LIN {X 0,Y 108.125,Z 394.279,A -85,B 0,C 180,E1 -26388.966,E2 -26388.966} C_VEL
LIN {X 0,Y 112.21,Z 392.494,A -85,B 0,C 180,E1 -26396.004,E2 -26396.004} C_VEL
LIN {X 0,Y 114.934,Z 391.013,A -85,B 0,C 180,E1 -26399.287,E2 -26399.287} C_VEL
LIN {X 0,Y 119.605,Z 388.035,A -85,B 0,C 180,E1 -26403.933,E2 -26403.933} C_VEL
LIN {X 0,Y 126.884,Z 382.493,A -85,B 0,C 180,E1 -26409.567,E2 -26409.567} C_VEL
LIN {X 0,Y 134.394,Z 376.043,A -85,B 0,C 180,E1 -26413.86,E2 -26413.86} C_VEL
LIN {X 0,Y 141.43,Z 369.031,A -85,B 0,C 180,E1 -26417.136,E2 -26417.136} C_VEL
LIN {X 0,Y 148.869,Z 360.421,A -85,B 0,C 180,E1 -26420.1,E2 -26420.1} C_VEL
LIN {X 0,Y 151.521,Z 356.993,A -85,B 0,C 180,E1 -26421.065,E2 -26421.065} C_VEL
LIN {X 0,Y 154.305,Z 352.873,A -85,B 0,C 180,E1 -26422.25,E2 -26422.25} C_VEL
LIN {X 0,Y 157.695,Z 346.05,A -85,B 0,C 180,E1 -26424.594,E2 -26424.594} C_VEL
LIN {X 0,Y 160.885,Z 338.836,A -85,B 0,C 180,E1 -26426.75,E2 -26426.75} C_VEL
LIN {X 0,Y 163.243,Z 334.049,A -85,B 0,C 180,E1 -26427.636,E2 -26427.636} C_VEL
LIN {X 0,Y 168.407,Z 323.305,A -85,B 0,C 180,E1 -26428.817,E2 -26428.817} C_VEL
LIN {X 0,Y 172.662,Z 312.36,A -85,B 0,C 180,E1 -26429.673,E2 -26429.673} C_VEL
LIN {X 0,Y 176.386,Z 299.563,A -85,B 0,C 180,E1 -26430.418,E2 -26430.418} C_VEL
LIN {X 0,Y 179.004,Z 285.601,A -85,B 0,C 180,E1 -26430.963,E2 -26430.963} C_VEL
LIN {X 0,Y 179.557,Z 281.011,A -85,B 0,C 180,E1 -26431.149,E2 -26431.149} C_VEL
LIN {X 0,Y 178.226,Z 276.107,A -85,B 0,C 180,E1 -26433.713,E2 -26433.713} C_VEL
LIN {X 0,Y 177.2,Z 272.643,A -85,B 0,C 180,E1 -26436.252,E2 -26436.252} C_VEL
LIN {X 0,Y 176.323,Z 269.621,A -85,B 0,C 180,E1 -26439.283,E2 -26439.283} C_VEL
LIN {X 0,Y 175.677,Z 268.759,A -85,B 0,C 180,E1 -26443.768,E2 -26443.768} C_VEL
LIN {X 0,Y 176.5,Z 269.439,A -85,B 0,C 180,E1 -26449.627,E2 -26449.627} C_VEL
LIN {X 0,Y 177.757,Z 272.493,A -85,B 0,C 180,E1 -26453.188,E2 -26453.188} C_VEL
LIN {X 0,Y 179.592,Z 277.069,A -85,B 0,C 180,E1 -26456.689,E2 -26456.689} C_VEL
LIN {X 0,Y 179.895,Z 277.95,A -85,B 0,C 180,E1 -26457.192,E2 -26457.192} C_VEL
LIN {X 0,Y 177.766,Z 291.915,A -85,B 0,C 180,E1 -26457.679,E2 -26457.679} C_VEL
LIN {X 0,Y 174.451,Z 305.114,A -85,B 0,C 180,E1 -26458.412,E2 -26458.412} C_VEL
LIN {X 0,Y 170.441,Z 316.764,A -85,B 0,C 180,E1 -26459.359,E2 -26459.359} C_VEL
LIN {X 0,Y 165.172,Z 328.692,A -85,B 0,C 180,E1 -26460.698,E2 -26460.698} C_VEL
LIN {X 0,Y 159.012,Z 339.73,A -85,B 0,C 180,E1 -26462.356,E2 -26462.356} C_VEL
LIN {X 0,Y 152.408,Z 349.556,A -85,B 0,C 180,E1 -26464.299,E2 -26464.299} C_VEL
LIN {X 0,Y 145.085,Z 358.755,A -85,B 0,C 180,E1 -26466.765,E2 -26466.765} C_VEL
LIN {X 0,Y 137.182,Z 367.074,A -85,B 0,C 180,E1 -26469.864,E2 -26469.864} C_VEL
LIN {X 0,Y 129.973,Z 373.591,A -85,B 0,C 180,E1 -26473.265,E2 -26473.265} C_VEL
LIN {X 0,Y 124.361,Z 378.031,A -85,B 0,C 180,E1 -26476.414,E2 -26476.414} C_VEL
LIN {X 0,Y 117.458,Z 382.716,A -85,B 0,C 180,E1 -26481.039,E2 -26481.039} C_VEL
LIN {X 0,Y 110.517,Z 386.589,A -85,B 0,C 180,E1 -26487.09,E2 -26487.09} C_VEL
LIN {X 0,Y 106.415,Z 388.343,A -85,B 0,C 180,E1 -26491.894,E2 -26491.894} C_VEL
LIN {X 0,Y 102.395,Z 389.462,A -85,B 0,C 180,E1 -26498.15,E2 -26498.15} C_VEL
LIN {X 0,Y 99.483,Z 389.45,A -85,B 0,C 180,E1 -26505.052,E2 -26505.052} C_VEL
LIN {X 0,Y 97.861,Z 388.225,A -85,B 0,C 180,E1 -26512.184,E2 -26512.184} C_VEL
LIN {X 0,Y 97.493,Z 385.556,A -85,B 0,C 180,E1 -26519.889,E2 -26519.889} C_VEL
LIN {X 0,Y 98.329,Z 382.149,A -85,B 0,C 180,E1 -26526.375,E2 -26526.375} C_VEL
LIN {X 0,Y 100.113,Z 376.767,A -85,B 0,C 180,E1 -26533.692,E2 -26533.692} C_VEL
LIN {X 0,Y 102.685,Z 370.212,A -85,B 0,C 180,E1 -26540.148,E2 -26540.148} C_VEL
LIN {X 0,Y 106.375,Z 361.911,A -85,B 0,C 180,E1 -26546.212,E2 -26546.212} C_VEL
LIN {X 0,Y 110.108,Z 353.345,A -85,B 0,C 180,E1 -26550.914,E2 -26550.914} C_VEL
LIN {X 0,Y 114.038,Z 343.881,A -85,B 0,C 180,E1 -26554.861,E2 -26554.861} C_VEL
LIN {X 0,Y 118.414,Z 332.203,A -85,B 0,C 180,E1 -26558.533,E2 -26558.533} C_VEL
LIN {X 0,Y 122.062,Z 320.716,A -85,B 0,C 180,E1 -26561.194,E2 -26561.194} C_VEL
LIN {X 0,Y 125.332,Z 307.943,A -85,B 0,C 180,E1 -26563.374,E2 -26563.374} C_VEL
LIN {X 0,Y 127.759,Z 295.671,A -85,B 0,C 180,E1 -26564.841,E2 -26564.841} C_VEL
LIN {X 0,Y 129.611,Z 282.091,A -85,B 0,C 180,E1 -26565.854,E2 -26565.854} C_VEL
LIN {X 0,Y 132.721,Z 244.216,A -85,B 0,C 180,E1 -26567.762,E2 -26567.762} C_VEL
LIN {X 0,Y 126.635,Z 230.962,A -85,B 0,C 180,E1 -26571.189,E2 -26571.189} C_VEL
LIN {X 0,Y 120.083,Z 219.302,A -85,B 0,C 180,E1 -26575.232,E2 -26575.232} C_VEL
LIN {X 0,Y 116.054,Z 212.906,A -85,B 0,C 180,E1 -26577.99,E2 -26577.99} C_VEL
LIN {X 0,Y 112.722,Z 208.003,A -85,B 0,C 180,E1 -26580.499,E2 -26580.499} C_VEL
LIN {X 0,Y 110.582,Z 204.925,A -85,B 0,C 180,E1 -26582.238,E2 -26582.238} C_VEL
LIN {X 0,Y 107.998,Z 201.163,A -85,B 0,C 180,E1 -26584.514,E2 -26584.514} C_VEL
LIN {X 0,Y 105.595,Z 198.407,A -85,B 0,C 180,E1 -26586.744,E2 -26586.744} C_VEL
LIN {X 0,Y 104.678,Z 196.46,A -85,B 0,C 180,E1 -26587.788,E2 -26587.788} C_VEL
LIN {X 0,Y 102.258,Z 194.671,A -85,B 0,C 180,E1 -26590.208,E2 -26590.208} C_VEL
LIN {X 0,Y 100.868,Z 192.174,A -85,B 0,C 180,E1 -26591.976,E2 -26591.976} C_VEL
LIN {X 0,Y 100.591,Z 190.918,A -85,B 0,C 180,E1 -26592.553,E2 -26592.553} C_VEL
LIN {X 0,Y 100.632,Z 190.886,A -85,B 0,C 180,E1 -26595.702,E2 -26595.702} C_VEL
LIN {X 0,Y 100.617,Z 190.928,A -85,B 0,C 180,E1 -26601.05,E2 -26601.05} C_VEL
LIN {X 0,Y 100.688,Z 190.926,A -85,B 0,C 180,E1 -26606.888,E2 -26606.888} C_VEL
LIN {X 0,Y 100.735,Z 190.921,A -85,B 0,C 180,E1 -26615.092,E2 -26615.092} C_VEL
LIN {X 0,Y 100.782,Z 190.926,A -85,B 0,C 180,E1 -26619.594,E2 -26619.594} C_VEL
LIN {X 0,Y 101.126,Z 190.879,A -85,B 0,C 180,E1 -26627.966,E2 -26627.966} C_VEL
LIN {X 0,Y 101.229,Z 190.864,A -85,B 0,C 180,E1 -26632.018,E2 -26632.018} C_VEL
LIN {X 0,Y 101.827,Z 190.796,A -85,B 0,C 180,E1 -26640,E2 -26640} C_VEL
LIN {X 0,Y 101.221,Z 190.81,A -85,B 0,C 180,E1 -26647.982,E2 -26647.982} C_VEL
LIN {X 0,Y 100.973,Z 190.908,A -85,B 0,C 180,E1 -26654.182,E2 -26654.182} C_VEL
LIN {X 0,Y 100.895,Z 190.939,A -85,B 0,C 180,E1 -26655.432,E2 -26655.432} C_VEL
LIN {X 0,Y 101.676,Z 193.498,A -85,B 0,C 180,E1 -26656.618,E2 -26656.618} C_VEL
LIN {X 0,Y 103.54,Z 195.625,A -85,B 0,C 180,E1 -26658.681,E2 -26658.681} C_VEL
LIN {X 0,Y 104.952,Z 196.705,A -85,B 0,C 180,E1 -26660.071,E2 -26660.071} C_VEL
LIN {X 0,Y 106.785,Z 199.852,A -85,B 0,C 180,E1 -26661.982,E2 -26661.982} C_VEL
LIN {X 0,Y 108.619,Z 201.926,A -85,B 0,C 180,E1 -26663.626,E2 -26663.626} C_VEL
LIN {X 0,Y 111.232,Z 205.605,A -85,B 0,C 180,E1 -26665.864,E2 -26665.864} C_VEL
LIN {X 0,Y 116.524,Z 213.662,A -85,B 0,C 180,E1 -26669.931,E2 -26669.931} C_VEL
LIN {X 0,Y 122.986,Z 224.722,A -85,B 0,C 180,E1 -26674.235,E2 -26674.235} C_VEL
LIN {X 0,Y 127.867,Z 237.066,A -85,B 0,C 180,E1 -26677.417,E2 -26677.417} C_VEL
LIN {X 0,Y 132.368,Z 250.803,A -85,B 0,C 180,E1 -26680.206,E2 -26680.206} C_VEL
LIN {X 0,Y 129.045,Z 291.011,A -85,B 0,C 180,E1 -26682.278,E2 -26682.278} C_VEL
LIN {X 0,Y 126.907,Z 304.794,A -85,B 0,C 180,E1 -26683.462,E2 -26683.462} C_VEL
LIN {X 0,Y 123.943,Z 317.866,A -85,B 0,C 180,E1 -26685.15,E2 -26685.15} C_VEL
LIN {X 0,Y 120.552,Z 329.623,A -85,B 0,C 180,E1 -26687.334,E2 -26687.334} C_VEL
LIN {X 0,Y 116.497,Z 340.955,A -85,B 0,C 180,E1 -26690.134,E2 -26690.134} C_VEL
LIN {X 0,Y 112.958,Z 350.224,A -85,B 0,C 180,E1 -26693.212,E2 -26693.212} C_VEL
LIN {X 0,Y 109.225,Z 359.151,A -85,B 0,C 180,E1 -26697.022,E2 -26697.022} C_VEL
LIN {X 0,Y 105.259,Z 368.2,A -85,B 0,C 180,E1 -26702.136,E2 -26702.136} C_VEL
LIN {X 0,Y 102.065,Z 375.68,A -85,B 0,C 180,E1 -26707.746,E2 -26707.746} C_VEL
LIN {X 0,Y 99.806,Z 381.655,A -85,B 0,C 180,E1 -26713.64,E2 -26713.64} C_VEL
LIN {X 0,Y 98.544,Z 386.342,A -85,B 0,C 180,E1 -26719.73,E2 -26719.73} C_VEL
LIN {X 0,Y 98.097,Z 389.865,A -85,B 0,C 180,E1 -26725.892,E2 -26725.892} C_VEL
LIN {X 0,Y 98.185,Z 391.63,A -85,B 0,C 180,E1 -26730,E2 -26730} C_VEL
LIN {X 0,Y 98.047,Z 392.911,A -85,B 0,C 180,E1 -26734.111,E2 -26734.111} C_VEL
LIN {X 0,Y 98.878,Z 394.315,A -85,B 0,C 180,E1 -26742.312,E2 -26742.312} C_VEL
LIN {X 0,Y 99.917,Z 394.448,A -85,B 0,C 180,E1 -26746.341,E2 -26746.341} C_VEL
LIN {X 0,Y 103.36,Z 393.535,A -85,B 0,C 180,E1 -26754.078,E2 -26754.078} C_VEL
LIN {X 0,Y 108.773,Z 391.142,A -85,B 0,C 180,E1 -26761.124,E2 -26761.124} C_VEL
LIN {X 0,Y 113.794,Z 388.276,A -85,B 0,C 180,E1 -26765.925,E2 -26765.925} C_VEL
LIN {X 0,Y 119.475,Z 384.449,A -85,B 0,C 180,E1 -26770.321,E2 -26770.321} C_VEL
LIN {X 0,Y 125.943,Z 379.569,A -85,B 0,C 180,E1 -26774.23,E2 -26774.23} C_VEL
LIN {X 0,Y 133,Z 373.499,A -85,B 0,C 180,E1 -26777.714,E2 -26777.714} C_VEL
LIN {X 0,Y 140.554,Z 366.018,A -85,B 0,C 180,E1 -26780.809,E2 -26780.809} C_VEL
LIN {X 0,Y 148.504,Z 356.716,A -85,B 0,C 180,E1 -26783.566,E2 -26783.566} C_VEL
LIN {X 0,Y 156.12,Z 346.146,A -85,B 0,C 180,E1 -26785.811,E2 -26785.811} C_VEL
LIN {X 0,Y 162.557,Z 335.356,A -85,B 0,C 180,E1 -26787.466,E2 -26787.466} C_VEL
LIN {X 0,Y 163.243,Z 334.049,A -85,B 0,C 180,E1 -26787.636,E2 -26787.636} C_VEL
LIN {X 0,Y 165.524,Z 329.129,A -85,B 0,C 180,E1 -26788.451,E2 -26788.451} C_VEL
LIN {X 0,Y 168.292,Z 321.034,A -85,B 0,C 180,E1 -26790.189,E2 -26790.189} C_VEL
LIN {X 0,Y 170.727,Z 312.64,A -85,B 0,C 180,E1 -26791.73,E2 -26791.73} C_VEL
LIN {X 0,Y 172.343,Z 307.228,A -85,B 0,C 180,E1 -26792.26,E2 -26792.26} C_VEL
LIN {X 0,Y 175.702,Z 294.291,A -85,B 0,C 180,E1 -26792.872,E2 -26792.872} C_VEL
LIN {X 0,Y 177.27,Z 284.962,A -85,B 0,C 180,E1 -26793.217,E2 -26793.217} C_VEL
LIN {X 0,Y 176.285,Z 280.832,A -85,B 0,C 180,E1 -26795.757,E2 -26795.757} C_VEL
LIN {X 0,Y 175.735,Z 278.755,A -85,B 0,C 180,E1 -26797.474,E2 -26797.474} C_VEL
LIN {X 0,Y 175.269,Z 276.666,A -85,B 0,C 180,E1 -26799.459,E2 -26799.459} C_VEL
LIN {X 0,Y 174.683,Z 275.807,A -85,B 0,C 180,E1 -26803.643,E2 -26803.643} C_VEL
LIN {X 0,Y 175.322,Z 276.316,A -85,B 0,C 180,E1 -26808.998,E2 -26808.998} C_VEL
LIN {X 0,Y 175.628,Z 277.049,A -85,B 0,C 180,E1 -26810.183,E2 -26810.183} C_VEL
LIN {X 0,Y 176.419,Z 279.164,A -85,B 0,C 180,E1 -26812.512,E2 -26812.512} C_VEL
LIN {X 0,Y 177.554,Z 282.414,A -85,B 0,C 180,E1 -26815.131,E2 -26815.131} C_VEL
LIN {X 0,Y 174.975,Z 296.276,A -85,B 0,C 180,E1 -26815.655,E2 -26815.655} C_VEL
LIN {X 0,Y 171.545,Z 308.409,A -85,B 0,C 180,E1 -26816.363,E2 -26816.363} C_VEL
LIN {X 0,Y 167.054,Z 320.181,A -85,B 0,C 180,E1 -26817.365,E2 -26817.365} C_VEL
LIN {X 0,Y 161.692,Z 331.242,A -85,B 0,C 180,E1 -26818.631,E2 -26818.631} C_VEL
LIN {X 0,Y 155.383,Z 341.816,A -85,B 0,C 180,E1 -26820.226,E2 -26820.226} C_VEL
LIN {X 0,Y 148.569,Z 351.277,A -85,B 0,C 180,E1 -26822.112,E2 -26822.112} C_VEL
LIN {X 0,Y 140.996,Z 360.079,A -85,B 0,C 180,E1 -26824.502,E2 -26824.502} C_VEL
LIN {X 0,Y 132.912,Z 368.07,A -85,B 0,C 180,E1 -26827.502,E2 -26827.502} C_VEL
LIN {X 0,Y 125.263,Z 374.531,A -85,B 0,C 180,E1 -26830.93,E2 -26830.93} C_VEL
LIN {X 0,Y 116.755,Z 380.534,A -85,B 0,C 180,E1 -26835.608,E2 -26835.608} C_VEL
LIN {X 0,Y 109.129,Z 384.917,A -85,B 0,C 180,E1 -26840.962,E2 -26840.962} C_VEL
LIN {X 0,Y 102.63,Z 387.879,A -85,B 0,C 180,E1 -26847.097,E2 -26847.097} C_VEL
LIN {X 0,Y 98.989,Z 389.066,A -85,B 0,C 180,E1 -26851.572,E2 -26851.572} C_VEL
LIN {X 0,Y 95.957,Z 389.717,A -85,B 0,C 180,E1 -26856.326,E2 -26856.326} C_VEL
LIN {X 0,Y 92.977,Z 389.674,A -85,B 0,C 180,E1 -26862.867,E2 -26862.867} C_VEL
LIN {X 0,Y 90.997,Z 388.498,A -85,B 0,C 180,E1 -26870.564,E2 -26870.564} C_VEL
LIN {X 0,Y 90.369,Z 385.903,A -85,B 0,C 180,E1 -26878.812,E2 -26878.812} C_VEL
LIN {X 0,Y 91.383,Z 381.663,A -85,B 0,C 180,E1 -26887.385,E2 -26887.385} C_VEL
LIN {X 0,Y 93.216,Z 376.45,A -85,B 0,C 180,E1 -26894.697,E2 -26894.697} C_VEL
LIN {X 0,Y 96.009,Z 369.75,A -85,B 0,C 180,E1 -26901.581,E2 -26901.581} C_VEL
LIN {X 0,Y 99.299,Z 362.731,A -85,B 0,C 180,E1 -26907.018,E2 -26907.018} C_VEL
LIN {X 0,Y 103.183,Z 354.412,A -85,B 0,C 180,E1 -26911.952,E2 -26911.952} C_VEL
LIN {X 0,Y 107.386,Z 344.875,A -85,B 0,C 180,E1 -26916.222,E2 -26916.222} C_VEL
LIN {X 0,Y 111.876,Z 333.675,A -85,B 0,C 180,E1 -26919.948,E2 -26919.948} C_VEL
LIN {X 0,Y 115.91,Z 321.695,A -85,B 0,C 180,E1 -26922.914,E2 -26922.914} C_VEL
LIN {X 0,Y 119.303,Z 309.175,A -85,B 0,C 180,E1 -26925.154,E2 -26925.154} C_VEL
LIN {X 0,Y 122.094,Z 295.787,A -85,B 0,C 180,E1 -26926.819,E2 -26926.819} C_VEL
LIN {X 0,Y 124.033,Z 282.402,A -85,B 0,C 180,E1 -26927.821,E2 -26927.821} C_VEL
LIN {X 0,Y 127.2,Z 246.744,A -85,B 0,C 180,E1 -26929.618,E2 -26929.618} C_VEL
LIN {X 0,Y 122.027,Z 234.996,A -85,B 0,C 180,E1 -26932.852,E2 -26932.852} C_VEL
LIN {X 0,Y 115.732,Z 223.611,A -85,B 0,C 180,E1 -26937.054,E2 -26937.054} C_VEL
LIN {X 0,Y 112.142,Z 217.735,A -85,B 0,C 180,E1 -26939.769,E2 -26939.769} C_VEL
LIN {X 0,Y 109.294,Z 213.404,A -85,B 0,C 180,E1 -26942.096,E2 -26942.096} C_VEL
LIN {X 0,Y 105.067,Z 207.132,A -85,B 0,C 180,E1 -26945.974,E2 -26945.974} C_VEL
LIN {X 0,Y 102.472,Z 203.798,A -85,B 0,C 180,E1 -26948.646,E2 -26948.646} C_VEL
LIN {X 0,Y 101.623,Z 202.536,A -85,B 0,C 180,E1 -26949.605,E2 -26949.605} C_VEL
LIN {X 0,Y 99.259,Z 200.05,A -85,B 0,C 180,E1 -26952.351,E2 -26952.351} C_VEL
LIN {X 0,Y 98,Z 197.473,A -85,B 0,C 180,E1 -26954.181,E2 -26954.181} C_VEL
LIN {X 0,Y 95.181,Z 195.541,A -85,B 0,C 180,E1 -26958.117,E2 -26958.117} C_VEL
LIN {X 0,Y 93.895,Z 193.116,A -85,B 0,C 180,E1 -26960.523,E2 -26960.523} C_VEL
LIN {X 0,Y 93.565,Z 191.809,A -85,B 0,C 180,E1 -26961.476,E2 -26961.476} C_VEL
LIN {X 0,Y 93.576,Z 191.809,A -85,B 0,C 180,E1 -26968.282,E2 -26968.282} C_VEL
LIN {X 0,Y 93.644,Z 191.809,A -85,B 0,C 180,E1 -26974.238,E2 -26974.238} C_VEL
LIN {X 0,Y 93.654,Z 191.801,A -85,B 0,C 180,E1 -26977.962,E2 -26977.962} C_VEL
LIN {X 0,Y 94.016,Z 191.757,A -85,B 0,C 180,E1 -26987.04,E2 -26987.04} C_VEL
LIN {X 0,Y 94.16,Z 191.749,A -85,B 0,C 180,E1 -26991.415,E2 -26991.415} C_VEL
LIN {X 0,Y 94.756,Z 191.675,A -85,B 0,C 180,E1 -27000,E2 -27000} C_VEL
LIN {X 0,Y 94.162,Z 191.71,A -85,B 0,C 180,E1 -27007.101,E2 -27007.101} C_VEL
LIN {X 0,Y 95.042,Z 194.419,A -85,B 0,C 180,E1 -27009.04,E2 -27009.04} C_VEL
LIN {X 0,Y 96.964,Z 196.611,A -85,B 0,C 180,E1 -27012.027,E2 -27012.027} C_VEL
LIN {X 0,Y 98.325,Z 197.699,A -85,B 0,C 180,E1 -27013.827,E2 -27013.827} C_VEL
LIN {X 0,Y 99.951,Z 200.763,A -85,B 0,C 180,E1 -27016.073,E2 -27016.073} C_VEL
LIN {X 0,Y 102.289,Z 203.059,A -85,B 0,C 180,E1 -27018.658,E2 -27018.658} C_VEL
LIN {X 0,Y 104.615,Z 206.547,A -85,B 0,C 180,E1 -27021.167,E2 -27021.167} C_VEL
LIN {X 0,Y 105.907,Z 208.364,A -85,B 0,C 180,E1 -27022.431,E2 -27022.431} C_VEL
LIN {X 0,Y 109.082,Z 213.08,A -85,B 0,C 180,E1 -27025.31,E2 -27025.31} C_VEL
LIN {X 0,Y 112.766,Z 218.729,A -85,B 0,C 180,E1 -27028.31,E2 -27028.31} C_VEL
LIN {X 0,Y 118.777,Z 229.384,A -85,B 0,C 180,E1 -27032.674,E2 -27032.674} C_VEL
LIN {X 0,Y 123.785,Z 242.908,A -85,B 0,C 180,E1 -27036.231,E2 -27036.231} C_VEL
LIN {X 0,Y 126.819,Z 252.699,A -85,B 0,C 180,E1 -27038.314,E2 -27038.314} C_VEL
LIN {X 0,Y 123.374,Z 291.507,A -85,B 0,C 180,E1 -27040.354,E2 -27040.354} C_VEL
LIN {X 0,Y 121.024,Z 305.612,A -85,B 0,C 180,E1 -27041.611,E2 -27041.611} C_VEL
LIN {X 0,Y 118.154,Z 317.664,A -85,B 0,C 180,E1 -27043.226,E2 -27043.226} C_VEL
LIN {X 0,Y 114.315,Z 330.197,A -85,B 0,C 180,E1 -27045.627,E2 -27045.627} C_VEL
LIN {X 0,Y 110.142,Z 341.412,A -85,B 0,C 180,E1 -27048.546,E2 -27048.546} C_VEL
LIN {X 0,Y 105.993,Z 351.595,A -85,B 0,C 180,E1 -27052.169,E2 -27052.169} C_VEL
LIN {X 0,Y 101.817,Z 360.761,A -85,B 0,C 180,E1 -27056.481,E2 -27056.481} C_VEL
LIN {X 0,Y 97.765,Z 369.727,A -85,B 0,C 180,E1 -27062.143,E2 -27062.143} C_VEL
LIN {X 0,Y 94.498,Z 376.849,A -85,B 0,C 180,E1 -27068.17,E2 -27068.17} C_VEL
LIN {X 0,Y 92.399,Z 382.527,A -85,B 0,C 180,E1 -27074.561,E2 -27074.561} C_VEL
LIN {X 0,Y 91.279,Z 386.953,A -85,B 0,C 180,E1 -27081.142,E2 -27081.142} C_VEL
LIN {X 0,Y 91.038,Z 389.269,A -85,B 0,C 180,E1 -27085.572,E2 -27085.572} C_VEL
LIN {X 0,Y 91.106,Z 391.134,A -85,B 0,C 180,E1 -27090,E2 -27090} C_VEL
LIN {X 0,Y 90.974,Z 392.5,A -85,B 0,C 180,E1 -27094.431,E2 -27094.431} C_VEL
LIN {X 0,Y 91.924,Z 394.021,A -85,B 0,C 180,E1 -27103.26,E2 -27103.26} C_VEL
LIN {X 0,Y 94.733,Z 394.063,A -85,B 0,C 180,E1 -27111.774,E2 -27111.774} C_VEL
LIN {X 0,Y 99.629,Z 392.559,A -85,B 0,C 180,E1 -27119.59,E2 -27119.59} C_VEL
LIN {X 0,Y 106.226,Z 389.545,A -85,B 0,C 180,E1 -27126.545,E2 -27126.545} C_VEL
LIN {X 0,Y 112.115,Z 386.174,A -85,B 0,C 180,E1 -27131.216,E2 -27131.216} C_VEL
LIN {X 0,Y 118.608,Z 381.859,A -85,B 0,C 180,E1 -27135.321,E2 -27135.321} C_VEL
LIN {X 0,Y 127.083,Z 375.376,A -85,B 0,C 180,E1 -27139.501,E2 -27139.501} C_VEL
LIN {X 0,Y 134.87,Z 368.333,A -85,B 0,C 180,E1 -27142.625,E2 -27142.625} C_VEL
LIN {X 0,Y 143.017,Z 359.679,A -85,B 0,C 180,E1 -27145.398,E2 -27145.398} C_VEL
LIN {X 0,Y 150.152,Z 350.876,A -85,B 0,C 180,E1 -27147.407,E2 -27147.407} C_VEL
LIN {X 0,Y 157.454,Z 340.096,A -85,B 0,C 180,E1 -27149.231,E2 -27149.231} C_VEL
LIN {X 0,Y 163.417,Z 329.334,A -85,B 0,C 180,E1 -27150.563,E2 -27150.563} C_VEL
LIN {X 0,Y 168.828,Z 317.198,A -85,B 0,C 180,E1 -27151.652,E2 -27151.652} C_VEL
LIN {X 0,Y 172.343,Z 307.228,A -85,B 0,C 180,E1 -27152.26,E2 -27152.26} C_VEL
LIN {X 0,Y 174.151,Z 300.463,A -85,B 0,C 180,E1 -27152.759,E2 -27152.759} C_VEL
LIN {X 0,Y 175.003,Z 295.302,A -85,B 0,C 180,E1 -27153.463,E2 -27153.463} C_VEL
LIN {X 0,Y 175.266,Z 291.94,A -85,B 0,C 180,E1 -27154.218,E2 -27154.218} C_VEL
LIN {X 0,Y 175.189,Z 289.141,A -85,B 0,C 180,E1 -27155.305,E2 -27155.305} C_VEL
LIN {X 0,Y 175.112,Z 288.691,A -85,B 0,C 180,E1 -27155.598,E2 -27155.598} C_VEL
LIN {X 0,Y 174.47,Z 285.533,A -85,B 0,C 180,E1 -27158.033,E2 -27158.033} C_VEL
LIN {X 0,Y 174.145,Z 283.561,A -85,B 0,C 180,E1 -27159.937,E2 -27159.937} C_VEL
LIN {X 0,Y 173.687,Z 282.83,A -85,B 0,C 180,E1 -27163.546,E2 -27163.546} C_VEL
LIN {X 0,Y 174.274,Z 283.343,A -85,B 0,C 180,E1 -27168.931,E2 -27168.931} C_VEL
LIN {X 0,Y 175.039,Z 285.885,A -85,B 0,C 180,E1 -27171.89,E2 -27171.89} C_VEL
LIN {X 0,Y 175.39,Z 287.202,A -85,B 0,C 180,E1 -27172.997,E2 -27172.997} C_VEL
LIN {X 0,Y 172.289,Z 300.871,A -85,B 0,C 180,E1 -27173.59,E2 -27173.59} C_VEL
LIN {X 0,Y 168.101,Z 313.557,A -85,B 0,C 180,E1 -27174.38,E2 -27174.38} C_VEL
LIN {X 0,Y 162.91,Z 325.379,A -85,B 0,C 180,E1 -27175.469,E2 -27175.469} C_VEL
LIN {X 0,Y 156.607,Z 336.769,A -85,B 0,C 180,E1 -27176.878,E2 -27176.878} C_VEL
LIN {X 0,Y 149.389,Z 347.396,A -85,B 0,C 180,E1 -27178.637,E2 -27178.637} C_VEL
LIN {X 0,Y 141.813,Z 356.544,A -85,B 0,C 180,E1 -27180.676,E2 -27180.676} C_VEL
LIN {X 0,Y 133.745,Z 364.769,A -85,B 0,C 180,E1 -27183.227,E2 -27183.227} C_VEL
LIN {X 0,Y 125.209,Z 372.119,A -85,B 0,C 180,E1 -27186.446,E2 -27186.446} C_VEL
LIN {X 0,Y 116.633,Z 378.279,A -85,B 0,C 180,E1 -27190.415,E2 -27190.415} C_VEL
LIN {X 0,Y 108.729,Z 382.997,A -85,B 0,C 180,E1 -27194.984,E2 -27194.984} C_VEL
LIN {X 0,Y 101.523,Z 386.463,A -85,B 0,C 180,E1 -27200.251,E2 -27200.251} C_VEL
LIN {X 0,Y 94.716,Z 388.937,A -85,B 0,C 180,E1 -27207.074,E2 -27207.074} C_VEL
LIN {X 0,Y 90.395,Z 389.851,A -85,B 0,C 180,E1 -27212.973,E2 -27212.973} C_VEL
LIN {X 0,Y 86.562,Z 389.891,A -85,B 0,C 180,E1 -27220.506,E2 -27220.506} C_VEL
LIN {X 0,Y 84.173,Z 388.752,A -85,B 0,C 180,E1 -27228.717,E2 -27228.717} C_VEL
LIN {X 0,Y 83.25,Z 386.217,A -85,B 0,C 180,E1 -27237.587,E2 -27237.587} C_VEL
LIN {X 0,Y 84.12,Z 382.083,A -85,B 0,C 180,E1 -27246.785,E2 -27246.785} C_VEL
LIN {X 0,Y 85.62,Z 377.986,A -85,B 0,C 180,E1 -27253.304,E2 -27253.304} C_VEL
LIN {X 0,Y 88.267,Z 371.716,A -85,B 0,C 180,E1 -27260.837,E2 -27260.837} C_VEL
LIN {X 0,Y 91.507,Z 365.051,A -85,B 0,C 180,E1 -27266.8,E2 -27266.8} C_VEL
LIN {X 0,Y 95.431,Z 357.204,A -85,B 0,C 180,E1 -27272.11,E2 -27272.11} C_VEL
LIN {X 0,Y 99.668,Z 348.221,A -85,B 0,C 180,E1 -27276.73,E2 -27276.73} C_VEL
LIN {X 0,Y 104.197,Z 337.919,A -85,B 0,C 180,E1 -27280.689,E2 -27280.689} C_VEL
LIN {X 0,Y 108.639,Z 326.279,A -85,B 0,C 180,E1 -27283.981,E2 -27283.981} C_VEL
LIN {X 0,Y 112.516,Z 313.785,A -85,B 0,C 180,E1 -27286.558,E2 -27286.558} C_VEL
LIN {X 0,Y 115.635,Z 301.034,A -85,B 0,C 180,E1 -27288.401,E2 -27288.401} C_VEL
LIN {X 0,Y 117.974,Z 287.454,A -85,B 0,C 180,E1 -27289.684,E2 -27289.684} C_VEL
LIN {X 0,Y 120.828,Z 259.224,A -85,B 0,C 180,E1 -27291.178,E2 -27291.178} C_VEL
LIN {X 0,Y 121.665,Z 248.784,A -85,B 0,C 180,E1 -27291.755,E2 -27291.755} C_VEL
LIN {X 0,Y 117.402,Z 238.926,A -85,B 0,C 180,E1 -27294.652,E2 -27294.652} C_VEL
LIN {X 0,Y 110.775,Z 226.511,A -85,B 0,C 180,E1 -27299.624,E2 -27299.624} C_VEL
LIN {X 0,Y 105.682,Z 218.384,A -85,B 0,C 180,E1 -27304.011,E2 -27304.011} C_VEL
LIN {X 0,Y 102.05,Z 212.89,A -85,B 0,C 180,E1 -27307.686,E2 -27307.686} C_VEL
LIN {X 0,Y 99.085,Z 208.732,A -85,B 0,C 180,E1 -27311.095,E2 -27311.095} C_VEL
LIN {X 0,Y 96.616,Z 205.773,A -85,B 0,C 180,E1 -27314.262,E2 -27314.262} C_VEL
LIN {X 0,Y 95.582,Z 203.923,A -85,B 0,C 180,E1 -27315.866,E2 -27315.866} C_VEL
LIN {X 0,Y 92.938,Z 201.582,A -85,B 0,C 180,E1 -27320.035,E2 -27320.035} C_VEL
LIN {X 0,Y 91.688,Z 198.792,A -85,B 0,C 180,E1 -27322.799,E2 -27322.799} C_VEL
LIN {X 0,Y 87.915,Z 196.06,A -85,B 0,C 180,E1 -27333.106,E2 -27333.106} C_VEL
LIN {X 0,Y 86.955,Z 194.171,A -85,B 0,C 180,E1 -27339.909,E2 -27339.909} C_VEL
LIN {X 0,Y 87.025,Z 193.205,A -85,B 0,C 180,E1 -27346.808,E2 -27346.808} C_VEL
LIN {X 0,Y 87.744,Z 194.827,A -85,B 0,C 180,E1 -27353.099,E2 -27353.099} C_VEL
LIN {X 0,Y 90.071,Z 197.179,A -85,B 0,C 180,E1 -27361.118,E2 -27361.118} C_VEL
LIN {X 0,Y 92.184,Z 198.642,A -85,B 0,C 180,E1 -27365.605,E2 -27365.605} C_VEL
LIN {X 0,Y 93.488,Z 201.529,A -85,B 0,C 180,E1 -27368.348,E2 -27368.348} C_VEL
LIN {X 0,Y 95.984,Z 204.127,A -85,B 0,C 180,E1 -27372.265,E2 -27372.265} C_VEL
LIN {X 0,Y 98.071,Z 207.567,A -85,B 0,C 180,E1 -27375.256,E2 -27375.256} C_VEL
LIN {X 0,Y 99.714,Z 209.296,A -85,B 0,C 180,E1 -27377.199,E2 -27377.199} C_VEL
LIN {X 0,Y 103.111,Z 214.452,A -85,B 0,C 180,E1 -27381.032,E2 -27381.032} C_VEL
LIN {X 0,Y 107.722,Z 221.521,A -85,B 0,C 180,E1 -27385.397,E2 -27385.397} C_VEL
LIN {X 0,Y 113.248,Z 231.423,A -85,B 0,C 180,E1 -27389.97,E2 -27389.97} C_VEL
LIN {X 0,Y 114.874,Z 234.857,A -85,B 0,C 180,E1 -27391.222,E2 -27391.222} C_VEL
LIN {X 0,Y 119.056,Z 246.618,A -85,B 0,C 180,E1 -27394.445,E2 -27394.445} C_VEL
LIN {X 0,Y 121.373,Z 254.383,A -85,B 0,C 180,E1 -27396.212,E2 -27396.212} C_VEL
LIN {X 0,Y 117.89,Z 291.693,A -85,B 0,C 180,E1 -27398.22,E2 -27398.22} C_VEL
LIN {X 0,Y 115.496,Z 305.398,A -85,B 0,C 180,E1 -27399.462,E2 -27399.462} C_VEL
LIN {X 0,Y 112.51,Z 317.461,A -85,B 0,C 180,E1 -27401.106,E2 -27401.106} C_VEL
LIN {X 0,Y 108.772,Z 329.207,A -85,B 0,C 180,E1 -27403.374,E2 -27403.374} C_VEL
LIN {X 0,Y 104.366,Z 340.559,A -85,B 0,C 180,E1 -27406.351,E2 -27406.351} C_VEL
LIN {X 0,Y 99.964,Z 350.894,A -85,B 0,C 180,E1 -27410.093,E2 -27410.093} C_VEL
LIN {X 0,Y 95.957,Z 359.331,A -85,B 0,C 180,E1 -27414.131,E2 -27414.131} C_VEL
LIN {X 0,Y 91.507,Z 368.49,A -85,B 0,C 180,E1 -27420.052,E2 -27420.052} C_VEL
LIN {X 0,Y 87.929,Z 375.828,A -85,B 0,C 180,E1 -27426.444,E2 -27426.444} C_VEL
LIN {X 0,Y 85.535,Z 381.689,A -85,B 0,C 180,E1 -27433.287,E2 -27433.287} C_VEL
LIN {X 0,Y 84.26,Z 386.263,A -85,B 0,C 180,E1 -27440.397,E2 -27440.397} C_VEL
LIN {X 0,Y 83.968,Z 388.648,A -85,B 0,C 180,E1 -27445.199,E2 -27445.199} C_VEL
LIN {X 0,Y 84.013,Z 390.577,A -85,B 0,C 180,E1 -27450,E2 -27450} C_VEL
LIN {X 0,Y 83.921,Z 392.044,A -85,B 0,C 180,E1 -27454.804,E2 -27454.804} C_VEL
LIN {X 0,Y 84.196,Z 393.086,A -85,B 0,C 180,E1 -27459.61,E2 -27459.61} C_VEL
LIN {X 0,Y 86.321,Z 393.996,A -85,B 0,C 180,E1 -27469.006,E2 -27469.006} C_VEL
LIN {X 0,Y 90.568,Z 393.445,A -85,B 0,C 180,E1 -27477.749,E2 -27477.749} C_VEL
LIN {X 0,Y 96.854,Z 391.362,A -85,B 0,C 180,E1 -27485.486,E2 -27485.486} C_VEL
LIN {X 0,Y 104.715,Z 387.73,A -85,B 0,C 180,E1 -27492.157,E2 -27492.157} C_VEL
LIN {X 0,Y 111.348,Z 383.885,A -85,B 0,C 180,E1 -27496.54,E2 -27496.54} C_VEL
LIN {X 0,Y 118.767,Z 378.967,A -85,B 0,C 180,E1 -27500.289,E2 -27500.289} C_VEL
LIN {X 0,Y 126.647,Z 372.882,A -85,B 0,C 180,E1 -27503.577,E2 -27503.577} C_VEL
LIN {X 0,Y 134.943,Z 365.386,A -85,B 0,C 180,E1 -27506.44,E2 -27506.44} C_VEL
LIN {X 0,Y 142.1,Z 357.795,A -85,B 0,C 180,E1 -27508.557,E2 -27508.557} C_VEL
LIN {X 0,Y 150.236,Z 347.57,A -85,B 0,C 180,E1 -27510.608,E2 -27510.608} C_VEL
LIN {X 0,Y 157.054,Z 337.268,A -85,B 0,C 180,E1 -27512.104,E2 -27512.104} C_VEL
LIN {X 0,Y 163.214,Z 325.907,A -85,B 0,C 180,E1 -27513.317,E2 -27513.317} C_VEL
LIN {X 0,Y 168.162,Z 314.449,A -85,B 0,C 180,E1 -27514.171,E2 -27514.171} C_VEL
LIN {X 0,Y 172.656,Z 300.541,A -85,B 0,C 180,E1 -27514.903,E2 -27514.903} C_VEL
LIN {X 0,Y 175.159,Z 289.078,A -85,B 0,C 180,E1 -27515.376,E2 -27515.376} C_VEL
LIN {X 0,Y 175.112,Z 288.691,A -85,B 0,C 180,E1 -27515.598,E2 -27515.598} C_VEL
LIN {X 0,Y 174.701,Z 287.528,A -85,B 0,C 180,E1 -27516.82,E2 -27516.82} C_VEL
LIN {X 0,Y 173.987,Z 287.033,A -85,B 0,C 180,E1 -27518.747,E2 -27518.747} C_VEL
LIN {X 0,Y 172.949,Z 288.207,A -85,B 0,C 180,E1 -27522.042,E2 -27522.042} C_VEL
LIN {X 0,Y 172.504,Z 289.527,A -85,B 0,C 180,E1 -27524.734,E2 -27524.734} C_VEL
LIN {X 0,Y 172.532,Z 289.863,A -85,B 0,C 180,E1 -27526.095,E2 -27526.095} C_VEL
LIN {X 0,Y 172.958,Z 290.433,A -85,B 0,C 180,E1 -27528.899,E2 -27528.899} C_VEL
LIN {X 0,Y 173.318,Z 292.045,A -85,B 0,C 180,E1 -27530.864,E2 -27530.864} C_VEL
LIN {X 0,Y 170.006,Z 304.609,A -85,B 0,C 180,E1 -27531.43,E2 -27531.43} C_VEL
LIN {X 0,Y 165.402,Z 317.07,A -85,B 0,C 180,E1 -27532.244,E2 -27532.244} C_VEL
LIN {X 0,Y 160.118,Z 328.143,A -85,B 0,C 180,E1 -27533.256,E2 -27533.256} C_VEL
LIN {X 0,Y 153.753,Z 338.86,A -85,B 0,C 180,E1 -27534.561,E2 -27534.561} C_VEL
LIN {X 0,Y 146.389,Z 348.94,A -85,B 0,C 180,E1 -27536.206,E2 -27536.206} C_VEL
LIN {X 0,Y 138.883,Z 357.512,A -85,B 0,C 180,E1 -27538.067,E2 -27538.067} C_VEL
LIN {X 0,Y 130.028,Z 366.062,A -85,B 0,C 180,E1 -27540.658,E2 -27540.658} C_VEL
LIN {X 0,Y 122.434,Z 372.227,A -85,B 0,C 180,E1 -27543.291,E2 -27543.291} C_VEL
LIN {X 0,Y 113.329,Z 378.452,A -85,B 0,C 180,E1 -27547.145,E2 -27547.145} C_VEL
LIN {X 0,Y 104.901,Z 383.156,A -85,B 0,C 180,E1 -27551.595,E2 -27551.595} C_VEL
LIN {X 0,Y 95.937,Z 387.095,A -85,B 0,C 180,E1 -27557.759,E2 -27557.759} C_VEL
LIN {X 0,Y 90.398,Z 388.891,A -85,B 0,C 180,E1 -27562.876,E2 -27562.876} C_VEL
LIN {X 0,Y 84.731,Z 390.053,A -85,B 0,C 180,E1 -27569.846,E2 -27569.846} C_VEL
LIN {X 0,Y 80.241,Z 390.096,A -85,B 0,C 180,E1 -27577.975,E2 -27577.975} C_VEL
LIN {X 0,Y 77.441,Z 388.995,A -85,B 0,C 180,E1 -27586.555,E2 -27586.555} C_VEL
LIN {X 0,Y 76.168,Z 386.445,A -85,B 0,C 180,E1 -27596.384,E2 -27596.384} C_VEL
LIN {X 0,Y 76.879,Z 382.495,A -85,B 0,C 180,E1 -27606.089,E2 -27606.089} C_VEL
LIN {X 0,Y 78.717,Z 377.648,A -85,B 0,C 180,E1 -27614.464,E2 -27614.464} C_VEL
LIN {X 0,Y 81.667,Z 371.194,A -85,B 0,C 180,E1 -27622.583,E2 -27622.583} C_VEL
LIN {X 0,Y 85.949,Z 362.986,A -85,B 0,C 180,E1 -27630,E2 -27630} C_VEL
LIN {X 0,Y 90.223,Z 354.908,A -85,B 0,C 180,E1 -27635.35,E2 -27635.35} C_VEL
LIN {X 0,Y 94.989,Z 345.218,A -85,B 0,C 180,E1 -27640.121,E2 -27640.121} C_VEL
LIN {X 0,Y 100.078,Z 333.692,A -85,B 0,C 180,E1 -27644.231,E2 -27644.231} C_VEL
LIN {X 0,Y 104.252,Z 322.519,A -85,B 0,C 180,E1 -27647.154,E2 -27647.154} C_VEL
LIN {X 0,Y 108.023,Z 310.119,A -85,B 0,C 180,E1 -27649.477,E2 -27649.477} C_VEL
LIN {X 0,Y 111.064,Z 296.92,A -85,B 0,C 180,E1 -27651.216,E2 -27651.216} C_VEL
LIN {X 0,Y 113.284,Z 283.141,A -85,B 0,C 180,E1 -27652.29,E2 -27652.29} C_VEL
LIN {X 0,Y 116.345,Z 250.985,A -85,B 0,C 180,E1 -27653.997,E2 -27653.997} C_VEL
LIN {X 0,Y 112.902,Z 242.907,A -85,B 0,C 180,E1 -27656.589,E2 -27656.589} C_VEL
LIN {X 0,Y 107.059,Z 231.495,A -85,B 0,C 180,E1 -27661.416,E2 -27661.416} C_VEL
LIN {X 0,Y 101.761,Z 222.571,A -85,B 0,C 180,E1 -27666.534,E2 -27666.534} C_VEL
LIN {X 0,Y 99.046,Z 218.531,A -85,B 0,C 180,E1 -27669.577,E2 -27669.577} C_VEL
LIN {X 0,Y 96.441,Z 214.783,A -85,B 0,C 180,E1 -27672.837,E2 -27672.837} C_VEL
LIN {X 0,Y 93.922,Z 211.195,A -85,B 0,C 180,E1 -27676.549,E2 -27676.549} C_VEL
LIN {X 0,Y 93.141,Z 210.193,A -85,B 0,C 180,E1 -27677.832,E2 -27677.832} C_VEL
LIN {X 0,Y 90.804,Z 207.57,A -85,B 0,C 180,E1 -27682.059,E2 -27682.059} C_VEL
LIN {X 0,Y 89.792,Z 205.437,A -85,B 0,C 180,E1 -27684.519,E2 -27684.519} C_VEL
LIN {X 0,Y 86.637,Z 202.809,A -85,B 0,C 180,E1 -27694.329,E2 -27694.329} C_VEL
LIN {X 0,Y 85.882,Z 200.68,A -85,B 0,C 180,E1 -27702.744,E2 -27702.744} C_VEL
LIN {X 0,Y 86.062,Z 200.414,A -85,B 0,C 180,E1 -27707.55,E2 -27707.55} C_VEL
LIN {X 0,Y 86.607,Z 201.767,A -85,B 0,C 180,E1 -27712.422,E2 -27712.422} C_VEL
LIN {X 0,Y 89.035,Z 204.313,A -85,B 0,C 180,E1 -27721.131,E2 -27721.131} C_VEL
LIN {X 0,Y 90.37,Z 205.403,A -85,B 0,C 180,E1 -27724.181,E2 -27724.181} C_VEL
LIN {X 0,Y 91.956,Z 208.429,A -85,B 0,C 180,E1 -27727.595,E2 -27727.595} C_VEL
LIN {X 0,Y 93.82,Z 210.6,A -85,B 0,C 180,E1 -27730.789,E2 -27730.789} C_VEL
LIN {X 0,Y 96.167,Z 214.277,A -85,B 0,C 180,E1 -27734.351,E2 -27734.351} C_VEL
LIN {X 0,Y 97.603,Z 216.197,A -85,B 0,C 180,E1 -27736.21,E2 -27736.21} C_VEL
LIN {X 0,Y 100.585,Z 220.831,A -85,B 0,C 180,E1 -27739.782,E2 -27739.782} C_VEL
LIN {X 0,Y 104.544,Z 227.267,A -85,B 0,C 180,E1 -27743.873,E2 -27743.873} C_VEL
LIN {X 0,Y 110.028,Z 237.557,A -85,B 0,C 180,E1 -27748.754,E2 -27748.754} C_VEL
LIN {X 0,Y 113.817,Z 248.394,A -85,B 0,C 180,E1 -27752.049,E2 -27752.049} C_VEL
LIN {X 0,Y 116.069,Z 256.166,A -85,B 0,C 180,E1 -27753.949,E2 -27753.949} C_VEL
LIN {X 0,Y 112.676,Z 290.844,A -85,B 0,C 180,E1 -27755.82,E2 -27755.82} C_VEL
LIN {X 0,Y 110.307,Z 304.229,A -85,B 0,C 180,E1 -27757.021,E2 -27757.021} C_VEL
LIN {X 0,Y 107.041,Z 317.088,A -85,B 0,C 180,E1 -27758.768,E2 -27758.768} C_VEL
LIN {X 0,Y 102.813,Z 329.636,A -85,B 0,C 180,E1 -27761.242,E2 -27761.242} C_VEL
LIN {X 0,Y 98.236,Z 340.873,A -85,B 0,C 180,E1 -27764.322,E2 -27764.322} C_VEL
LIN {X 0,Y 93.537,Z 351.219,A -85,B 0,C 180,E1 -27768.277,E2 -27768.277} C_VEL
LIN {X 0,Y 89.386,Z 359.443,A -85,B 0,C 180,E1 -27772.457,E2 -27772.457} C_VEL
LIN {X 0,Y 84.67,Z 368.547,A -85,B 0,C 180,E1 -27778.75,E2 -27778.75} C_VEL
LIN {X 0,Y 80.911,Z 375.841,A -85,B 0,C 180,E1 -27785.632,E2 -27785.632} C_VEL
LIN {X 0,Y 78.734,Z 380.752,A -85,B 0,C 180,E1 -27791.795,E2 -27791.795} C_VEL
LIN {X 0,Y 77.253,Z 385.495,A -85,B 0,C 180,E1 -27799.517,E2 -27799.517} C_VEL
LIN {X 0,Y 76.839,Z 389.067,A -85,B 0,C 180,E1 -27807.379,E2 -27807.379} C_VEL
LIN {X 0,Y 76.931,Z 390.016,A -85,B 0,C 180,E1 -27810,E2 -27810} C_VEL
LIN {X 0,Y 76.854,Z 391.55,A -85,B 0,C 180,E1 -27815.247,E2 -27815.247} C_VEL
LIN {X 0,Y 78.139,Z 393.427,A -85,B 0,C 180,E1 -27825.654,E2 -27825.654} C_VEL
LIN {X 0,Y 81.655,Z 393.739,A -85,B 0,C 180,E1 -27835.49,E2 -27835.49} C_VEL
LIN {X 0,Y 87.557,Z 392.609,A -85,B 0,C 180,E1 -27844.186,E2 -27844.186} C_VEL
LIN {X 0,Y 91.152,Z 391.484,A -85,B 0,C 180,E1 -27848.084,E2 -27848.084} C_VEL
LIN {X 0,Y 99.559,Z 388.005,A -85,B 0,C 180,E1 -27854.904,E2 -27854.904} C_VEL
LIN {X 0,Y 106.598,Z 384.342,A -85,B 0,C 180,E1 -27859.306,E2 -27859.306} C_VEL
LIN {X 0,Y 114.387,Z 379.625,A -85,B 0,C 180,E1 -27863.009,E2 -27863.009} C_VEL
LIN {X 0,Y 124.025,Z 372.633,A -85,B 0,C 180,E1 -27866.702,E2 -27866.702} C_VEL
LIN {X 0,Y 132.659,Z 365.125,A -85,B 0,C 180,E1 -27869.417,E2 -27869.417} C_VEL
LIN {X 0,Y 141.577,Z 355.805,A -85,B 0,C 180,E1 -27871.779,E2 -27871.779} C_VEL
LIN {X 0,Y 150.04,Z 345.251,A -85,B 0,C 180,E1 -27873.616,E2 -27873.616} C_VEL
LIN {X 0,Y 157.067,Z 334.477,A -85,B 0,C 180,E1 -27874.972,E2 -27874.972} C_VEL
LIN {X 0,Y 163.202,Z 322.834,A -85,B 0,C 180,E1 -27876.026,E2 -27876.026} C_VEL
LIN {X 0,Y 168.272,Z 310.63,A -85,B 0,C 180,E1 -27876.759,E2 -27876.759} C_VEL
LIN {X 0,Y 172.275,Z 297.221,A -85,B 0,C 180,E1 -27877.357,E2 -27877.357} C_VEL
LIN {X 0,Y 173.124,Z 293.578,A -85,B 0,C 180,E1 -27877.513,E2 -27877.513} C_VEL
LIN {X 0,Y 172.807,Z 290.439,A -85,B 0,C 180,E1 -27880.353,E2 -27880.353} C_VEL
LIN {X 0,Y 172.458,Z 289.83,A -85,B 0,C 180,E1 -27883.425,E2 -27883.425} C_VEL
LIN {X 0,Y 172.532,Z 289.863,A -85,B 0,C 180,E1 -27886.095,E2 -27886.095} C_VEL
LIN {X 0,Y 172.479,Z 290.829,A -85,B 0,C 180,E1 -27887.08,E2 -27887.08} C_VEL
LIN {X 0,Y 172.189,Z 292.909,A -85,B 0,C 180,E1 -27887.888,E2 -27887.888} C_VEL
LIN {X 0,Y 171.364,Z 296.969,A -85,B 0,C 180,E1 -27888.728,E2 -27888.728} C_VEL
LIN {X 0,Y 170.425,Z 300.602,A -85,B 0,C 180,E1 -27889.125,E2 -27889.125} C_VEL
LIN {X 0,Y 167.475,Z 309.652,A -85,B 0,C 180,E1 -27889.499,E2 -27889.499} C_VEL
LIN {X 0,Y 163.963,Z 318.171,A -85,B 0,C 180,E1 -27889.865,E2 -27889.865} C_VEL
LIN {X 0,Y 158.294,Z 329.536,A -85,B 0,C 180,E1 -27890.847,E2 -27890.847} C_VEL
LIN {X 0,Y 150.942,Z 341.153,A -85,B 0,C 180,E1 -27892.208,E2 -27892.208} C_VEL
LIN {X 0,Y 143.155,Z 351.176,A -85,B 0,C 180,E1 -27893.801,E2 -27893.801} C_VEL
LIN {X 0,Y 135.707,Z 359.159,A -85,B 0,C 180,E1 -27895.507,E2 -27895.507} C_VEL
LIN {X 0,Y 126.586,Z 367.348,A -85,B 0,C 180,E1 -27897.951,E2 -27897.951} C_VEL
LIN {X 0,Y 117.732,Z 373.963,A -85,B 0,C 180,E1 -27900.824,E2 -27900.824} C_VEL
LIN {X 0,Y 108.212,Z 379.875,A -85,B 0,C 180,E1 -27904.648,E2 -27904.648} C_VEL
LIN {X 0,Y 99.614,Z 384.2,A -85,B 0,C 180,E1 -27908.98,E2 -27908.98} C_VEL
LIN {X 0,Y 93.096,Z 386.819,A -85,B 0,C 180,E1 -27913.09,E2 -27913.09} C_VEL
LIN {X 0,Y 85.672,Z 389.093,A -85,B 0,C 180,E1 -27919.156,E2 -27919.156} C_VEL
LIN {X 0,Y 78.852,Z 390.316,A -85,B 0,C 180,E1 -27926.963,E2 -27926.963} C_VEL
LIN {X 0,Y 74.298,Z 390.319,A -85,B 0,C 180,E1 -27934.58,E2 -27934.58} C_VEL
LIN {X 0,Y 70.854,Z 389.228,A -85,B 0,C 180,E1 -27943.974,E2 -27943.974} C_VEL
LIN {X 0,Y 69.175,Z 386.821,A -85,B 0,C 180,E1 -27954.369,E2 -27954.369} C_VEL
LIN {X 0,Y 69.609,Z 382.85,A -85,B 0,C 180,E1 -27965.324,E2 -27965.324} C_VEL
LIN {X 0,Y 71.007,Z 379.147,A -85,B 0,C 180,E1 -27972.726,E2 -27972.726} C_VEL
LIN {X 0,Y 73.881,Z 373.034,A -85,B 0,C 180,E1 -27981.796,E2 -27981.796} C_VEL
LIN {X 0,Y 78.09,Z 365.319,A -85,B 0,C 180,E1 -27990,E2 -27990} C_VEL
LIN {X 0,Y 82.683,Z 357.254,A -85,B 0,C 180,E1 -27996.1,E2 -27996.1} C_VEL
LIN {X 0,Y 87.874,Z 347.45,A -85,B 0,C 180,E1 -28001.534,E2 -28001.534} C_VEL
LIN {X 0,Y 92.562,Z 337.82,A -85,B 0,C 180,E1 -28005.411,E2 -28005.411} C_VEL
LIN {X 0,Y 97.089,Z 327.113,A -85,B 0,C 180,E1 -28008.59,E2 -28008.59} C_VEL
LIN {X 0,Y 101.465,Z 314.421,A -85,B 0,C 180,E1 -28011.324,E2 -28011.324} C_VEL
LIN {X 0,Y 104.813,Z 302.012,A -85,B 0,C 180,E1 -28013.2,E2 -28013.2} C_VEL
LIN {X 0,Y 107.376,Z 288.894,A -85,B 0,C 180,E1 -28014.472,E2 -28014.472} C_VEL
LIN {X 0,Y 109.687,Z 269.033,A -85,B 0,C 180,E1 -28015.587,E2 -28015.587} C_VEL
LIN {X 0,Y 111.237,Z 253.447,A -85,B 0,C 180,E1 -28016.394,E2 -28016.394} C_VEL
LIN {X 0,Y 108.614,Z 247.068,A -85,B 0,C 180,E1 -28018.62,E2 -28018.62} C_VEL
LIN {X 0,Y 103.188,Z 236.062,A -85,B 0,C 180,E1 -28023.561,E2 -28023.561} C_VEL
LIN {X 0,Y 98.694,Z 228.08,A -85,B 0,C 180,E1 -28028.435,E2 -28028.435} C_VEL
LIN {X 0,Y 95.998,Z 223.963,A -85,B 0,C 180,E1 -28031.721,E2 -28031.721} C_VEL
LIN {X 0,Y 93.849,Z 220.719,A -85,B 0,C 180,E1 -28034.745,E2 -28034.745} C_VEL
LIN {X 0,Y 91.367,Z 216.819,A -85,B 0,C 180,E1 -28038.934,E2 -28038.934} C_VEL
LIN {X 0,Y 88.972,Z 213.969,A -85,B 0,C 180,E1 -28043.646,E2 -28043.646} C_VEL
LIN {X 0,Y 88.078,Z 212.16,A -85,B 0,C 180,E1 -28046.044,E2 -28046.044} C_VEL
LIN {X 0,Y 85.424,Z 209.616,A -85,B 0,C 180,E1 -28055.416,E2 -28055.416} C_VEL
LIN {X 0,Y 84.885,Z 207.702,A -85,B 0,C 180,E1 -28063.155,E2 -28063.155} C_VEL
LIN {X 0,Y 85.03,Z 207.39,A -85,B 0,C 180,E1 -28067.005,E2 -28067.005} C_VEL
LIN {X 0,Y 87.7,Z 211.198,A -85,B 0,C 180,E1 -28080.359,E2 -28080.359} C_VEL
LIN {X 0,Y 88.681,Z 212.152,A -85,B 0,C 180,E1 -28082.839,E2 -28082.839} C_VEL
LIN {X 0,Y 90.463,Z 215.443,A -85,B 0,C 180,E1 -28086.919,E2 -28086.919} C_VEL
LIN {X 0,Y 91.757,Z 217.063,A -85,B 0,C 180,E1 -28089.294,E2 -28089.294} C_VEL
LIN {X 0,Y 94.216,Z 220.909,A -85,B 0,C 180,E1 -28093.317,E2 -28093.317} C_VEL
LIN {X 0,Y 97.509,Z 226.166,A -85,B 0,C 180,E1 -28097.727,E2 -28097.727} C_VEL
LIN {X 0,Y 101.672,Z 233.439,A -85,B 0,C 180,E1 -28102.498,E2 -28102.498} C_VEL
LIN {X 0,Y 106.299,Z 242.702,A -85,B 0,C 180,E1 -28106.994,E2 -28106.994} C_VEL
LIN {X 0,Y 109.786,Z 253.743,A -85,B 0,C 180,E1 -28110.406,E2 -28110.406} C_VEL
LIN {X 0,Y 110.924,Z 257.847,A -85,B 0,C 180,E1 -28111.485,E2 -28111.485} C_VEL
LIN {X 0,Y 107.447,Z 291.47,A -85,B 0,C 180,E1 -28113.338,E2 -28113.338} C_VEL
LIN {X 0,Y 104.911,Z 304.834,A -85,B 0,C 180,E1 -28114.561,E2 -28114.561} C_VEL
LIN {X 0,Y 101.425,Z 317.618,A -85,B 0,C 180,E1 -28116.338,E2 -28116.338} C_VEL
LIN {X 0,Y 97.018,Z 330.012,A -85,B 0,C 180,E1 -28118.855,E2 -28118.855} C_VEL
LIN {X 0,Y 92.251,Z 341.16,A -85,B 0,C 180,E1 -28122.03,E2 -28122.03} C_VEL
LIN {X 0,Y 87.489,Z 351.004,A -85,B 0,C 180,E1 -28125.944,E2 -28125.944} C_VEL
LIN {X 0,Y 82.903,Z 359.553,A -85,B 0,C 180,E1 -28130.52,E2 -28130.52} C_VEL
LIN {X 0,Y 77.886,Z 368.604,A -85,B 0,C 180,E1 -28137.22,E2 -28137.22} C_VEL
LIN {X 0,Y 73.899,Z 375.847,A -85,B 0,C 180,E1 -28144.661,E2 -28144.661} C_VEL
LIN {X 0,Y 71.305,Z 381.606,A -85,B 0,C 180,E1 -28152.801,E2 -28152.801} C_VEL
LIN {X 0,Y 69.987,Z 386.096,A -85,B 0,C 180,E1 -28161.337,E2 -28161.337} C_VEL
LIN {X 0,Y 69.851,Z 389.447,A -85,B 0,C 180,E1 -28170,E2 -28170} C_VEL
LIN {X 0,Y 69.808,Z 391.044,A -85,B 0,C 180,E1 -28175.778,E2 -28175.778} C_VEL
LIN {X 0,Y 71.325,Z 393.066,A -85,B 0,C 180,E1 -28187.194,E2 -28187.194} C_VEL
LIN {X 0,Y 75.283,Z 393.577,A -85,B 0,C 180,E1 -28197.825,E2 -28197.825} C_VEL
LIN {X 0,Y 81.766,Z 392.59,A -85,B 0,C 180,E1 -28206.99,E2 -28206.99} C_VEL
LIN {X 0,Y 90.034,Z 390.147,A -85,B 0,C 180,E1 -28214.632,E2 -28214.632} C_VEL
LIN {X 0,Y 99.564,Z 386.074,A -85,B 0,C 180,E1 -28220.939,E2 -28220.939} C_VEL
LIN {X 0,Y 107.525,Z 381.888,A -85,B 0,C 180,E1 -28224.789,E2 -28224.789} C_VEL
LIN {X 0,Y 117.409,Z 375.599,A -85,B 0,C 180,E1 -28228.539,E2 -28228.539} C_VEL
LIN {X 0,Y 126.228,Z 368.862,A -85,B 0,C 180,E1 -28231.274,E2 -28231.274} C_VEL
LIN {X 0,Y 135.332,Z 360.543,A -85,B 0,C 180,E1 -28233.615,E2 -28233.615} C_VEL
LIN {X 0,Y 143.117,Z 352.078,A -85,B 0,C 180,E1 -28235.296,E2 -28235.296} C_VEL
LIN {X 0,Y 151.051,Z 341.744,A -85,B 0,C 180,E1 -28236.769,E2 -28236.769} C_VEL
LIN {X 0,Y 158.291,Z 330.178,A -85,B 0,C 180,E1 -28237.948,E2 -28237.948} C_VEL
LIN {X 0,Y 163.986,Z 318.675,A -85,B 0,C 180,E1 -28238.774,E2 -28238.774} C_VEL
LIN {X 0,Y 168.927,Z 305.777,A -85,B 0,C 180,E1 -28239.387,E2 -28239.387} C_VEL
LIN {X 0,Y 171.09,Z 298.363,A -85,B 0,C 180,E1 -28239.724,E2 -28239.724} C_VEL
LIN {X 0,Y 171.101,Z 297.245,A -85,B 0,C 180,E1 -28240.863,E2 -28240.863} C_VEL
LIN {X 0,Y 170.866,Z 296.764,A -85,B 0,C 180,E1 -28243.267,E2 -28243.267} C_VEL
LIN {X 0,Y 171.198,Z 297.043,A -85,B 0,C 180,E1 -28248.155,E2 -28248.155} C_VEL
LIN {X 0,Y 171.222,Z 297.479,A -85,B 0,C 180,E1 -28248.722,E2 -28248.722} C_VEL
LIN {X 0,Y 167.324,Z 309.909,A -85,B 0,C 180,E1 -28249.319,E2 -28249.319} C_VEL
LIN {X 0,Y 163.963,Z 318.171,A -85,B 0,C 180,E1 -28249.865,E2 -28249.865} C_VEL
LIN {X 0,Y 161.426,Z 323.502,A -85,B 0,C 180,E1 -28250.048,E2 -28250.048} C_VEL
LIN {X 0,Y 156.458,Z 332.084,A -85,B 0,C 180,E1 -28249.772,E2 -28249.772} C_VEL
LIN {X 0,Y 150.863,Z 340.219,A -85,B 0,C 180,E1 -28249.583,E2 -28249.583} C_VEL
LIN {X 0,Y 147.343,Z 344.836,A -85,B 0,C 180,E1 -28249.942,E2 -28249.942} C_VEL
LIN {X 0,Y 139.107,Z 354.447,A -85,B 0,C 180,E1 -28251.483,E2 -28251.483} C_VEL
LIN {X 0,Y 129.756,Z 363.496,A -85,B 0,C 180,E1 -28253.515,E2 -28253.515} C_VEL
LIN {X 0,Y 119.749,Z 371.366,A -85,B 0,C 180,E1 -28256.137,E2 -28256.137} C_VEL
LIN {X 0,Y 109.987,Z 377.662,A -85,B 0,C 180,E1 -28259.294,E2 -28259.294} C_VEL
LIN {X 0,Y 102.002,Z 381.898,A -85,B 0,C 180,E1 -28262.471,E2 -28262.471} C_VEL
LIN {X 0,Y 92.138,Z 386.103,A -85,B 0,C 180,E1 -28267.428,E2 -28267.428} C_VEL
LIN {X 0,Y 86.026,Z 388.103,A -85,B 0,C 180,E1 -28271.372,E2 -28271.372} C_VEL
LIN {X 0,Y 80.382,Z 389.533,A -85,B 0,C 180,E1 -28275.894,E2 -28275.894} C_VEL
LIN {X 0,Y 74.317,Z 390.466,A -85,B 0,C 180,E1 -28282.227,E2 -28282.227} C_VEL
LIN {X 0,Y 68.523,Z 390.531,A -85,B 0,C 180,E1 -28290.853,E2 -28290.853} C_VEL
LIN {X 0,Y 64.412,Z 389.457,A -85,B 0,C 180,E1 -28300.894,E2 -28300.894} C_VEL
LIN {X 0,Y 62.239,Z 387.103,A -85,B 0,C 180,E1 -28312.227,E2 -28312.227} C_VEL
LIN {X 0,Y 62.372,Z 383.198,A -85,B 0,C 180,E1 -28324.349,E2 -28324.349} C_VEL
LIN {X 0,Y 64.118,Z 378.749,A -85,B 0,C 180,E1 -28334.099,E2 -28334.099} C_VEL
LIN {X 0,Y 67.325,Z 372.496,A -85,B 0,C 180,E1 -28344.008,E2 -28344.008} C_VEL
LIN {X 0,Y 71.124,Z 366.023,A -85,B 0,C 180,E1 -28351.415,E2 -28351.415} C_VEL
LIN {X 0,Y 75.96,Z 358.107,A -85,B 0,C 180,E1 -28357.977,E2 -28357.977} C_VEL
LIN {X 0,Y 81.452,Z 348.415,A -85,B 0,C 180,E1 -28363.743,E2 -28363.743} C_VEL
LIN {X 0,Y 87.033,Z 337.687,A -85,B 0,C 180,E1 -28368.235,E2 -28368.235} C_VEL
LIN {X 0,Y 92.009,Z 326.381,A -85,B 0,C 180,E1 -28371.592,E2 -28371.592} C_VEL
LIN {X 0,Y 96.414,Z 314.134,A -85,B 0,C 180,E1 -28374.207,E2 -28374.207} C_VEL
LIN {X 0,Y 100.017,Z 301.2,A -85,B 0,C 180,E1 -28376.104,E2 -28376.104} C_VEL
LIN {X 0,Y 102.676,Z 287.654,A -85,B 0,C 180,E1 -28377.374,E2 -28377.374} C_VEL
LIN {X 0,Y 106.292,Z 256.03,A -85,B 0,C 180,E1 -28379.023,E2 -28379.023} C_VEL
LIN {X 0,Y 105.022,Z 252.473,A -85,B 0,C 180,E1 -28380.242,E2 -28380.242} C_VEL
LIN {X 0,Y 99.971,Z 241.622,A -85,B 0,C 180,E1 -28385.317,E2 -28385.317} C_VEL
LIN {X 0,Y 95.732,Z 233.66,A -85,B 0,C 180,E1 -28390.368,E2 -28390.368} C_VEL
LIN {X 0,Y 93.064,Z 229.302,A -85,B 0,C 180,E1 -28394.051,E2 -28394.051} C_VEL
LIN {X 0,Y 91.454,Z 226.708,A -85,B 0,C 180,E1 -28396.628,E2 -28396.628} C_VEL
LIN {X 0,Y 89.304,Z 223.209,A -85,B 0,C 180,E1 -28400.624,E2 -28400.624} C_VEL
LIN {X 0,Y 87.155,Z 220.213,A -85,B 0,C 180,E1 -28405.464,E2 -28405.464} C_VEL
LIN {X 0,Y 86.504,Z 218.888,A -85,B 0,C 180,E1 -28407.435,E2 -28407.435} C_VEL
LIN {X 0,Y 83.961,Z 215.614,A -85,B 0,C 180,E1 -28419.481,E2 -28419.481} C_VEL
LIN {X 0,Y 83.95,Z 214.456,A -85,B 0,C 180,E1 -28425.454,E2 -28425.454} C_VEL
LIN {X 0,Y 84.091,Z 214.733,A -85,B 0,C 180,E1 -28428.176,E2 -28428.176} C_VEL
LIN {X 0,Y 86.935,Z 218.55,A -85,B 0,C 180,E1 -28441.085,E2 -28441.085} C_VEL
LIN {X 0,Y 88.855,Z 222.212,A -85,B 0,C 180,E1 -28445.945,E2 -28445.945} C_VEL
LIN {X 0,Y 89.764,Z 223.498,A -85,B 0,C 180,E1 -28447.735,E2 -28447.735} C_VEL
LIN {X 0,Y 92.835,Z 228.651,A -85,B 0,C 180,E1 -28453.127,E2 -28453.127} C_VEL
LIN {X 0,Y 95.986,Z 234.103,A -85,B 0,C 180,E1 -28457.523,E2 -28457.523} C_VEL
LIN {X 0,Y 99.136,Z 240.262,A -85,B 0,C 180,E1 -28461.375,E2 -28461.375} C_VEL
LIN {X 0,Y 102.494,Z 247.545,A -85,B 0,C 180,E1 -28464.995,E2 -28464.995} C_VEL
LIN {X 0,Y 105.737,Z 258.587,A -85,B 0,C 180,E1 -28468.507,E2 -28468.507} C_VEL
LIN {X 0,Y 106.002,Z 260.206,A -85,B 0,C 180,E1 -28468.864,E2 -28468.864} C_VEL
LIN {X 0,Y 102.548,Z 291.286,A -85,B 0,C 180,E1 -28470.535,E2 -28470.535} C_VEL
LIN {X 0,Y 99.898,Z 304.707,A -85,B 0,C 180,E1 -28471.757,E2 -28471.757} C_VEL
LIN {X 0,Y 96.364,Z 317.161,A -85,B 0,C 180,E1 -28473.471,E2 -28473.471} C_VEL
LIN {X 0,Y 92.072,Z 328.81,A -85,B 0,C 180,E1 -28475.804,E2 -28475.804} C_VEL
LIN {X 0,Y 87.026,Z 340.117,A -85,B 0,C 180,E1 -28478.987,E2 -28478.987} C_VEL
LIN {X 0,Y 81.805,Z 350.4,A -85,B 0,C 180,E1 -28483.096,E2 -28483.096} C_VEL
LIN {X 0,Y 76.527,Z 359.621,A -85,B 0,C 180,E1 -28488.255,E2 -28488.255} C_VEL
LIN {X 0,Y 71.187,Z 368.618,A -85,B 0,C 180,E1 -28495.412,E2 -28495.412} C_VEL
LIN {X 0,Y 66.905,Z 375.798,A -85,B 0,C 180,E1 -28503.484,E2 -28503.484} C_VEL
LIN {X 0,Y 64.519,Z 380.649,A -85,B 0,C 180,E1 -28510.926,E2 -28510.926} C_VEL
LIN {X 0,Y 62.986,Z 385.314,A -85,B 0,C 180,E1 -28520.365,E2 -28520.365} C_VEL
LIN {X 0,Y 62.791,Z 388.812,A -85,B 0,C 180,E1 -28530,E2 -28530} C_VEL
LIN {X 0,Y 62.748,Z 390.526,A -85,B 0,C 180,E1 -28536.431,E2 -28536.431} C_VEL
LIN {X 0,Y 64.55,Z 392.691,A -85,B 0,C 180,E1 -28549.065,E2 -28549.065} C_VEL
LIN {X 0,Y 69.06,Z 393.383,A -85,B 0,C 180,E1 -28560.587,E2 -28560.587} C_VEL
LIN {X 0,Y 76.191,Z 392.585,A -85,B 0,C 180,E1 -28570.218,E2 -28570.218} C_VEL
LIN {X 0,Y 85.118,Z 390.3,A -85,B 0,C 180,E1 -28577.998,E2 -28577.998} C_VEL
LIN {X 0,Y 90.62,Z 388.385,A -85,B 0,C 180,E1 -28581.652,E2 -28581.652} C_VEL
LIN {X 0,Y 100.754,Z 383.899,A -85,B 0,C 180,E1 -28586.831,E2 -28586.831} C_VEL
LIN {X 0,Y 109.404,Z 379.203,A -85,B 0,C 180,E1 -28590.139,E2 -28590.139} C_VEL
LIN {X 0,Y 119.911,Z 372.249,A -85,B 0,C 180,E1 -28593.357,E2 -28593.357} C_VEL
LIN {X 0,Y 129.209,Z 364.783,A -85,B 0,C 180,E1 -28595.655,E2 -28595.655} C_VEL
LIN {X 0,Y 138.748,Z 355.486,A -85,B 0,C 180,E1 -28597.582,E2 -28597.582} C_VEL
LIN {X 0,Y 147.634,Z 344.988,A -85,B 0,C 180,E1 -28599.106,E2 -28599.106} C_VEL
LIN {X 0,Y 155,Z 334.3,A -85,B 0,C 180,E1 -28600.196,E2 -28600.196} C_VEL
LIN {X 0,Y 161.609,Z 322.32,A -85,B 0,C 180,E1 -28601.062,E2 -28601.062} C_VEL
LIN {X 0,Y 166.766,Z 310.369,A -85,B 0,C 180,E1 -28601.611,E2 -28601.611} C_VEL
LIN {X 0,Y 168.427,Z 305.609,A -85,B 0,C 180,E1 -28601.807,E2 -28601.807} C_VEL
LIN {X 0,Y 168.954,Z 303.73,A -85,B 0,C 180,E1 -28602.448,E2 -28602.448} C_VEL
LIN {X 0,Y 168.984,Z 303.586,A -85,B 0,C 180,E1 -28606.397,E2 -28606.397} C_VEL
LIN {X 0,Y 168.627,Z 304.761,A -85,B 0,C 180,E1 -28606.635,E2 -28606.635} C_VEL
LIN {X 0,Y 164.201,Z 316.383,A -85,B 0,C 180,E1 -28607.235,E2 -28607.235} C_VEL
LIN {X 0,Y 157.971,Z 328.907,A -85,B 0,C 180,E1 -28608.172,E2 -28608.172} C_VEL
LIN {X 0,Y 151.231,Z 339.594,A -85,B 0,C 180,E1 -28609.287,E2 -28609.287} C_VEL
LIN {X 0,Y 147.343,Z 344.836,A -85,B 0,C 180,E1 -28609.942,E2 -28609.942} C_VEL
LIN {X 0,Y 143.597,Z 349.382,A -85,B 0,C 180,E1 -28610.359,E2 -28610.359} C_VEL
LIN {X 0,Y 136.694,Z 356.577,A -85,B 0,C 180,E1 -28610.391,E2 -28610.391} C_VEL
LIN {X 0,Y 129.354,Z 363.127,A -85,B 0,C 180,E1 -28610.509,E2 -28610.509} C_VEL
LIN {X 0,Y 124.956,Z 366.677,A -85,B 0,C 180,E1 -28611.123,E2 -28611.123} C_VEL
LIN {X 0,Y 114.893,Z 373.815,A -85,B 0,C 180,E1 -28613.572,E2 -28613.572} C_VEL
LIN {X 0,Y 105.633,Z 379.212,A -85,B 0,C 180,E1 -28616.373,E2 -28616.373} C_VEL
LIN {X 0,Y 95.989,Z 383.748,A -85,B 0,C 180,E1 -28620,E2 -28620} C_VEL
LIN {X 0,Y 84.741,Z 387.744,A -85,B 0,C 180,E1 -28625.6,E2 -28625.6} C_VEL
LIN {X 0,Y 77.556,Z 389.512,A -85,B 0,C 180,E1 -28630.442,E2 -28630.442} C_VEL
LIN {X 0,Y 69.715,Z 390.676,A -85,B 0,C 180,E1 -28637.604,E2 -28637.604} C_VEL
LIN {X 0,Y 62.942,Z 390.732,A -85,B 0,C 180,E1 -28646.713,E2 -28646.713} C_VEL
LIN {X 0,Y 58.193,Z 389.672,A -85,B 0,C 180,E1 -28657.147,E2 -28657.147} C_VEL
LIN {X 0,Y 55.279,Z 387.124,A -85,B 0,C 180,E1 -28670.528,E2 -28670.528} C_VEL
LIN {X 0,Y 55.131,Z 383.522,A -85,B 0,C 180,E1 -28683.171,E2 -28683.171} C_VEL
LIN {X 0,Y 56.391,Z 380.207,A -85,B 0,C 180,E1 -28691.846,E2 -28691.846} C_VEL
LIN {X 0,Y 58.52,Z 375.968,A -85,B 0,C 180,E1 -28700.295,E2 -28700.295} C_VEL
LIN {X 0,Y 62.452,Z 369.424,A -85,B 0,C 180,E1 -28710,E2 -28710} C_VEL
LIN {X 0,Y 67.169,Z 362.219,A -85,B 0,C 180,E1 -28717.515,E2 -28717.515} C_VEL
LIN {X 0,Y 72.251,Z 354.307,A -85,B 0,C 180,E1 -28723.41,E2 -28723.41} C_VEL
LIN {X 0,Y 78.414,Z 343.747,A -85,B 0,C 180,E1 -28728.959,E2 -28728.959} C_VEL
LIN {X 0,Y 83.913,Z 333.027,A -85,B 0,C 180,E1 -28732.884,E2 -28732.884} C_VEL
LIN {X 0,Y 88.752,Z 321.699,A -85,B 0,C 180,E1 -28735.819,E2 -28735.819} C_VEL
LIN {X 0,Y 93.093,Z 308.982,A -85,B 0,C 180,E1 -28738.154,E2 -28738.154} C_VEL
LIN {X 0,Y 96.256,Z 296.734,A -85,B 0,C 180,E1 -28739.678,E2 -28739.678} C_VEL
LIN {X 0,Y 98.733,Z 282.763,A -85,B 0,C 180,E1 -28740.687,E2 -28740.687} C_VEL
LIN {X 0,Y 101.43,Z 257.71,A -85,B 0,C 180,E1 -28742.038,E2 -28742.038} C_VEL
LIN {X 0,Y 96.622,Z 246.631,A -85,B 0,C 180,E1 -28747.485,E2 -28747.485} C_VEL
LIN {X 0,Y 92.551,Z 238.628,A -85,B 0,C 180,E1 -28752.906,E2 -28752.906} C_VEL
LIN {X 0,Y 89.48,Z 233.174,A -85,B 0,C 180,E1 -28758.018,E2 -28758.018} C_VEL
LIN {X 0,Y 87.32,Z 229.558,A -85,B 0,C 180,E1 -28762.377,E2 -28762.377} C_VEL
LIN {X 0,Y 85.299,Z 226.178,A -85,B 0,C 180,E1 -28767.793,E2 -28767.793} C_VEL
LIN {X 0,Y 84.791,Z 225.484,A -85,B 0,C 180,E1 -28769.49,E2 -28769.49} C_VEL
LIN {X 0,Y 82.904,Z 221.726,A -85,B 0,C 180,E1 -28784.007,E2 -28784.007} C_VEL
LIN {X 0,Y 83.036,Z 221.651,A -85,B 0,C 180,E1 -28787.356,E2 -28787.356} C_VEL
LIN {X 0,Y 85.349,Z 225.19,A -85,B 0,C 180,E1 -28799.557,E2 -28799.557} C_VEL
LIN {X 0,Y 87.288,Z 228.995,A -85,B 0,C 180,E1 -28804.976,E2 -28804.976} C_VEL
LIN {X 0,Y 90.449,Z 234.656,A -85,B 0,C 180,E1 -28811.277,E2 -28811.277} C_VEL
LIN {X 0,Y 93.45,Z 240.376,A -85,B 0,C 180,E1 -28815.977,E2 -28815.977} C_VEL
LIN {X 0,Y 96.45,Z 246.573,A -85,B 0,C 180,E1 -28819.942,E2 -28819.942} C_VEL
LIN {X 0,Y 98.781,Z 252.323,A -85,B 0,C 180,E1 -28822.802,E2 -28822.802} C_VEL
LIN {X 0,Y 101.217,Z 261.373,A -85,B 0,C 180,E1 -28825.857,E2 -28825.857} C_VEL
LIN {X 0,Y 97.919,Z 290.657,A -85,B 0,C 180,E1 -28827.467,E2 -28827.467} C_VEL
LIN {X 0,Y 95.12,Z 304.31,A -85,B 0,C 180,E1 -28828.67,E2 -28828.67} C_VEL
LIN {X 0,Y 91.58,Z 316.435,A -85,B 0,C 180,E1 -28830.305,E2 -28830.305} C_VEL
LIN {X 0,Y 86.74,Z 328.989,A -85,B 0,C 180,E1 -28832.793,E2 -28832.793} C_VEL
LIN {X 0,Y 81.442,Z 340.231,A -85,B 0,C 180,E1 -28836,E2 -28836} C_VEL
LIN {X 0,Y 75.913,Z 350.442,A -85,B 0,C 180,E1 -28840.205,E2 -28840.205} C_VEL
LIN {X 0,Y 70.288,Z 359.619,A -85,B 0,C 180,E1 -28845.579,E2 -28845.579} C_VEL
LIN {X 0,Y 64.558,Z 368.584,A -85,B 0,C 180,E1 -28853.219,E2 -28853.219} C_VEL
LIN {X 0,Y 59.971,Z 375.727,A -85,B 0,C 180,E1 -28862.046,E2 -28862.046} C_VEL
LIN {X 0,Y 57.037,Z 381.409,A -85,B 0,C 180,E1 -28872.058,E2 -28872.058} C_VEL
LIN {X 0,Y 55.742,Z 385.84,A -85,B 0,C 180,E1 -28882.757,E2 -28882.757} C_VEL
LIN {X 0,Y 55.719,Z 388.147,A -85,B 0,C 180,E1 -28890,E2 -28890} C_VEL
LIN {X 0,Y 55.716,Z 389.954,A -85,B 0,C 180,E1 -28897.247,E2 -28897.247} C_VEL
LIN {X 0,Y 56.402,Z 391.339,A -85,B 0,C 180,E1 -28904.431,E2 -28904.431} C_VEL
LIN {X 0,Y 60.107,Z 392.907,A -85,B 0,C 180,E1 -28917.885,E2 -28917.885} C_VEL
LIN {X 0,Y 66.708,Z 393.037,A -85,B 0,C 180,E1 -28929.208,E2 -28929.208} C_VEL
LIN {X 0,Y 75.525,Z 391.699,A -85,B 0,C 180,E1 -28938.112,E2 -28938.112} C_VEL
LIN {X 0,Y 85.788,Z 388.844,A -85,B 0,C 180,E1 -28945.008,E2 -28945.008} C_VEL
LIN {X 0,Y 94.135,Z 385.676,A -85,B 0,C 180,E1 -28949.158,E2 -28949.158} C_VEL
LIN {X 0,Y 103.042,Z 381.514,A -85,B 0,C 180,E1 -28952.459,E2 -28952.459} C_VEL
LIN {X 0,Y 112.255,Z 376.257,A -85,B 0,C 180,E1 -28955.206,E2 -28955.206} C_VEL
LIN {X 0,Y 121.709,Z 369.753,A -85,B 0,C 180,E1 -28957.506,E2 -28957.506} C_VEL
LIN {X 0,Y 131.349,Z 361.791,A -85,B 0,C 180,E1 -28959.451,E2 -28959.451} C_VEL
LIN {X 0,Y 139.523,Z 353.714,A -85,B 0,C 180,E1 -28960.817,E2 -28960.817} C_VEL
LIN {X 0,Y 147.79,Z 343.929,A -85,B 0,C 180,E1 -28962.006,E2 -28962.006} C_VEL
LIN {X 0,Y 155.302,Z 332.983,A -85,B 0,C 180,E1 -28962.939,E2 -28962.939} C_VEL
LIN {X 0,Y 162.021,Z 320.743,A -85,B 0,C 180,E1 -28963.669,E2 -28963.669} C_VEL
LIN {X 0,Y 165.84,Z 311.969,A -85,B 0,C 180,E1 -28963.998,E2 -28963.998} C_VEL
LIN {X 0,Y 166.515,Z 310.247,A -85,B 0,C 180,E1 -28964.252,E2 -28964.252} C_VEL
LIN {X 0,Y 166.248,Z 310.892,A -85,B 0,C 180,E1 -28964.465,E2 -28964.465} C_VEL
LIN {X 0,Y 161.19,Z 322.318,A -85,B 0,C 180,E1 -28965.121,E2 -28965.121} C_VEL
LIN {X 0,Y 154.837,Z 333.594,A -85,B 0,C 180,E1 -28965.98,E2 -28965.98} C_VEL
LIN {X 0,Y 147.875,Z 343.583,A -85,B 0,C 180,E1 -28966.983,E2 -28966.983} C_VEL
LIN {X 0,Y 139.294,Z 353.601,A -85,B 0,C 180,E1 -28968.357,E2 -28968.357} C_VEL
LIN {X 0,Y 130.237,Z 362.296,A -85,B 0,C 180,E1 -28970.01,E2 -28970.01} C_VEL
LIN {X 0,Y 124.956,Z 366.677,A -85,B 0,C 180,E1 -28971.123,E2 -28971.123} C_VEL
LIN {X 0,Y 120.382,Z 370.094,A -85,B 0,C 180,E1 -28971.841,E2 -28971.841} C_VEL
LIN {X 0,Y 112.027,Z 375.332,A -85,B 0,C 180,E1 -28972.375,E2 -28972.375} C_VEL
LIN {X 0,Y 103.35,Z 379.877,A -85,B 0,C 180,E1 -28973.102,E2 -28973.102} C_VEL
LIN {X 0,Y 98.318,Z 382.168,A -85,B 0,C 180,E1 -28974.242,E2 -28974.242} C_VEL
LIN {X 0,Y 87.898,Z 386.193,A -85,B 0,C 180,E1 -28978.125,E2 -28978.125} C_VEL
LIN {X 0,Y 77.448,Z 389.112,A -85,B 0,C 180,E1 -28983.433,E2 -28983.433} C_VEL
LIN {X 0,Y 70.94,Z 390.299,A -85,B 0,C 180,E1 -28987.814,E2 -28987.814} C_VEL
LIN {X 0,Y 64.929,Z 390.953,A -85,B 0,C 180,E1 -28993.049,E2 -28993.049} C_VEL
LIN {X 0,Y 58.133,Z 390.953,A -85,B 0,C 180,E1 -29001.266,E2 -29001.266} C_VEL
LIN {X 0,Y 51.433,Z 389.549,A -85,B 0,C 180,E1 -29014.928,E2 -29014.928} C_VEL
LIN {X 0,Y 48.659,Z 387.588,A -85,B 0,C 180,E1 -29026.235,E2 -29026.235} C_VEL
LIN {X 0,Y 47.928,Z 383.813,A -85,B 0,C 180,E1 -29041.622,E2 -29041.622} C_VEL
LIN {X 0,Y 49.473,Z 379.777,A -85,B 0,C 180,E1 -29053.494,E2 -29053.494} C_VEL
LIN {X 0,Y 53.008,Z 373.655,A -85,B 0,C 180,E1 -29066.199,E2 -29066.199} C_VEL
LIN {X 0,Y 58.354,Z 365.954,A -85,B 0,C 180,E1 -29076.917,E2 -29076.917} C_VEL
LIN {X 0,Y 64.553,Z 357.196,A -85,B 0,C 180,E1 -29084.833,E2 -29084.833} C_VEL
LIN {X 0,Y 71.107,Z 347.079,A -85,B 0,C 180,E1 -29090.995,E2 -29090.995} C_VEL
LIN {X 0,Y 77.252,Z 336.239,A -85,B 0,C 180,E1 -29095.377,E2 -29095.377} C_VEL
LIN {X 0,Y 82.651,Z 324.915,A -85,B 0,C 180,E1 -29098.575,E2 -29098.575} C_VEL
LIN {X 0,Y 87.177,Z 313.174,A -85,B 0,C 180,E1 -29100.927,E2 -29100.927} C_VEL
LIN {X 0,Y 91.033,Z 299.942,A -85,B 0,C 180,E1 -29102.712,E2 -29102.712} C_VEL
LIN {X 0,Y 93.729,Z 287.047,A -85,B 0,C 180,E1 -29103.78,E2 -29103.78} C_VEL
LIN {X 0,Y 96.931,Z 260.534,A -85,B 0,C 180,E1 -29105.135,E2 -29105.135} C_VEL
LIN {X 0,Y 93.079,Z 251.025,A -85,B 0,C 180,E1 -29110.158,E2 -29110.158} C_VEL
LIN {X 0,Y 89.135,Z 242.648,A -85,B 0,C 180,E1 -29116.405,E2 -29116.405} C_VEL
LIN {X 0,Y 86.637,Z 238.188,A -85,B 0,C 180,E1 -29121.28,E2 -29121.28} C_VEL
LIN {X 0,Y 85.489,Z 235.975,A -85,B 0,C 180,E1 -29124.05,E2 -29124.05} C_VEL
LIN {X 0,Y 83.69,Z 232.495,A -85,B 0,C 180,E1 -29129.744,E2 -29129.744} C_VEL
LIN {X 0,Y 81.91,Z 228.747,A -85,B 0,C 180,E1 -29144.447,E2 -29144.447} C_VEL
LIN {X 0,Y 82.018,Z 228.752,A -85,B 0,C 180,E1 -29147.196,E2 -29147.196} C_VEL
LIN {X 0,Y 83.886,Z 231.966,A -85,B 0,C 180,E1 -29158.226,E2 -29158.226} C_VEL
LIN {X 0,Y 85.998,Z 236.552,A -85,B 0,C 180,E1 -29164.687,E2 -29164.687} C_VEL
LIN {X 0,Y 88.438,Z 241.212,A -85,B 0,C 180,E1 -29169.872,E2 -29169.872} C_VEL
LIN {X 0,Y 91.555,Z 247.772,A -85,B 0,C 180,E1 -29175.211,E2 -29175.211} C_VEL
LIN {X 0,Y 94.931,Z 256.004,A -85,B 0,C 180,E1 -29180.001,E2 -29180.001} C_VEL
LIN {X 0,Y 96.771,Z 263.415,A -85,B 0,C 180,E1 -29182.732,E2 -29182.732} C_VEL
LIN {X 0,Y 93.409,Z 291.041,A -85,B 0,C 180,E1 -29184.181,E2 -29184.181} C_VEL
LIN {X 0,Y 90.43,Z 304.82,A -85,B 0,C 180,E1 -29185.382,E2 -29185.382} C_VEL
LIN {X 0,Y 86.737,Z 316.731,A -85,B 0,C 180,E1 -29186.964,E2 -29186.964} C_VEL
LIN {X 0,Y 81.67,Z 329.162,A -85,B 0,C 180,E1 -29189.39,E2 -29189.39} C_VEL
LIN {X 0,Y 76.112,Z 340.345,A -85,B 0,C 180,E1 -29192.585,E2 -29192.585} C_VEL
LIN {X 0,Y 70.103,Z 350.73,A -85,B 0,C 180,E1 -29196.978,E2 -29196.978} C_VEL
LIN {X 0,Y 64.227,Z 359.616,A -85,B 0,C 180,E1 -29202.386,E2 -29202.386} C_VEL
LIN {X 0,Y 58.032,Z 368.547,A -85,B 0,C 180,E1 -29210.52,E2 -29210.52} C_VEL
LIN {X 0,Y 53.078,Z 375.643,A -85,B 0,C 180,E1 -29220.229,E2 -29220.229} C_VEL
LIN {X 0,Y 49.578,Z 382.1,A -85,B 0,C 180,E1 -29233.53,E2 -29233.53} C_VEL
LIN {X 0,Y 48.568,Z 386.3,A -85,B 0,C 180,E1 -29245.851,E2 -29245.851} C_VEL
LIN {X 0,Y 48.631,Z 387.456,A -85,B 0,C 180,E1 -29250,E2 -29250} C_VEL
LIN {X 0,Y 48.708,Z 389.335,A -85,B 0,C 180,E1 -29258.296,E2 -29258.296} C_VEL
LIN {X 0,Y 51.313,Z 391.894,A -85,B 0,C 180,E1 -29274.261,E2 -29274.261} C_VEL
LIN {X 0,Y 57.259,Z 392.914,A -85,B 0,C 180,E1 -29287.858,E2 -29287.858} C_VEL
LIN {X 0,Y 65.951,Z 392.49,A -85,B 0,C 180,E1 -29298.241,E2 -29298.241} C_VEL
LIN {X 0,Y 76.338,Z 390.629,A -85,B 0,C 180,E1 -29305.954,E2 -29305.954} C_VEL
LIN {X 0,Y 87.734,Z 387.195,A -85,B 0,C 180,E1 -29311.784,E2 -29311.784} C_VEL
LIN {X 0,Y 96.857,Z 383.546,A -85,B 0,C 180,E1 -29315.097,E2 -29315.097} C_VEL
LIN {X 0,Y 106.28,Z 378.895,A -85,B 0,C 180,E1 -29317.788,E2 -29317.788} C_VEL
LIN {X 0,Y 117.57,Z 371.991,A -85,B 0,C 180,E1 -29320.305,E2 -29320.305} C_VEL
LIN {X 0,Y 127.398,Z 364.603,A -85,B 0,C 180,E1 -29322.104,E2 -29322.104} C_VEL
LIN {X 0,Y 135.728,Z 357.097,A -85,B 0,C 180,E1 -29323.323,E2 -29323.323} C_VEL
LIN {X 0,Y 143.127,Z 349.215,A -85,B 0,C 180,E1 -29324.277,E2 -29324.277} C_VEL
LIN {X 0,Y 143.729,Z 348.512,A -85,B 0,C 180,E1 -29324.711,E2 -29324.711} C_VEL
LIN {X 0,Y 135.918,Z 356.798,A -85,B 0,C 180,E1 -29325.819,E2 -29325.819} C_VEL
LIN {X 0,Y 126.418,Z 365.143,A -85,B 0,C 180,E1 -29327.376,E2 -29327.376} C_VEL
LIN {X 0,Y 115.764,Z 372.795,A -85,B 0,C 180,E1 -29329.506,E2 -29329.506} C_VEL
LIN {X 0,Y 104.659,Z 379.182,A -85,B 0,C 180,E1 -29332.282,E2 -29332.282} C_VEL
LIN {X 0,Y 98.318,Z 382.168,A -85,B 0,C 180,E1 -29334.242,E2 -29334.242} C_VEL
LIN {X 0,Y 93.213,Z 384.253,A -85,B 0,C 180,E1 -29335.547,E2 -29335.547} C_VEL
LIN {X 0,Y 84.02,Z 387.259,A -85,B 0,C 180,E1 -29337.01,E2 -29337.01} C_VEL
LIN {X 0,Y 74.752,Z 389.482,A -85,B 0,C 180,E1 -29338.928,E2 -29338.928} C_VEL
LIN {X 0,Y 69.643,Z 390.282,A -85,B 0,C 180,E1 -29341.168,E2 -29341.168} C_VEL
LIN {X 0,Y 62.158,Z 391.113,A -85,B 0,C 180,E1 -29346.492,E2 -29346.492} C_VEL
LIN {X 0,Y 53.688,Z 391.161,A -85,B 0,C 180,E1 -29355.178,E2 -29355.178} C_VEL
LIN {X 0,Y 46.787,Z 390.091,A -85,B 0,C 180,E1 -29366.785,E2 -29366.785} C_VEL
LIN {X 0,Y 42.152,Z 387.814,A -85,B 0,C 180,E1 -29381.83,E2 -29381.83} C_VEL
LIN {X 0,Y 40.75,Z 384.088,A -85,B 0,C 180,E1 -29399.581,E2 -29399.581} C_VEL
LIN {X 0,Y 42.405,Z 379.694,A -85,B 0,C 180,E1 -29414.644,E2 -29414.644} C_VEL
LIN {X 0,Y 45.912,Z 374.179,A -85,B 0,C 180,E1 -29427.807,E2 -29427.807} C_VEL
LIN {X 0,Y 51.668,Z 366.564,A -85,B 0,C 180,E1 -29439.789,E2 -29439.789} C_VEL
LIN {X 0,Y 57.672,Z 358.847,A -85,B 0,C 180,E1 -29447.518,E2 -29447.518} C_VEL
LIN {X 0,Y 64.634,Z 348.957,A -85,B 0,C 180,E1 -29454.064,E2 -29454.064} C_VEL
LIN {X 0,Y 71.326,Z 338.208,A -85,B 0,C 180,E1 -29458.708,E2 -29458.708} C_VEL
LIN {X 0,Y 77.539,Z 326.121,A -85,B 0,C 180,E1 -29462.175,E2 -29462.175} C_VEL
LIN {X 0,Y 82.689,Z 313.593,A -85,B 0,C 180,E1 -29464.638,E2 -29464.638} C_VEL
LIN {X 0,Y 86.79,Z 300.184,A -85,B 0,C 180,E1 -29466.379,E2 -29466.379} C_VEL
LIN {X 0,Y 89.717,Z 286.612,A -85,B 0,C 180,E1 -29467.436,E2 -29467.436} C_VEL
LIN {X 0,Y 92.663,Z 263.165,A -85,B 0,C 180,E1 -29468.566,E2 -29468.566} C_VEL
LIN {X 0,Y 89.503,Z 254.94,A -85,B 0,C 180,E1 -29473.42,E2 -29473.42} C_VEL
LIN {X 0,Y 86.711,Z 248.427,A -85,B 0,C 180,E1 -29478.638,E2 -29478.638} C_VEL
LIN {X 0,Y 84.738,Z 244.541,A -85,B 0,C 180,E1 -29483.001,E2 -29483.001} C_VEL
LIN {X 0,Y 83.715,Z 242.398,A -85,B 0,C 180,E1 -29485.835,E2 -29485.835} C_VEL
LIN {X 0,Y 82.221,Z 239.236,A -85,B 0,C 180,E1 -29491.289,E2 -29491.289} C_VEL
LIN {X 0,Y 80.923,Z 235.747,A -85,B 0,C 180,E1 -29504.897,E2 -29504.897} C_VEL
LIN {X 0,Y 80.986,Z 235.786,A -85,B 0,C 180,E1 -29506.687,E2 -29506.687} C_VEL
LIN {X 0,Y 82.443,Z 238.633,A -85,B 0,C 180,E1 -29516.711,E2 -29516.711} C_VEL
LIN {X 0,Y 84.188,Z 242.997,A -85,B 0,C 180,E1 -29522.991,E2 -29522.991} C_VEL
LIN {X 0,Y 86.185,Z 247.177,A -85,B 0,C 180,E1 -29527.802,E2 -29527.802} C_VEL
LIN {X 0,Y 88.982,Z 253.721,A -85,B 0,C 180,E1 -29533.279,E2 -29533.279} C_VEL
LIN {X 0,Y 91.558,Z 260.8,A -85,B 0,C 180,E1 -29537.511,E2 -29537.511} C_VEL
LIN {X 0,Y 92.585,Z 265.303,A -85,B 0,C 180,E1 -29539.271,E2 -29539.271} C_VEL
LIN {X 0,Y 89.318,Z 290.873,A -85,B 0,C 180,E1 -29540.553,E2 -29540.553} C_VEL
LIN {X 0,Y 86.129,Z 304.958,A -85,B 0,C 180,E1 -29541.712,E2 -29541.712} C_VEL
LIN {X 0,Y 82.218,Z 316.906,A -85,B 0,C 180,E1 -29543.232,E2 -29543.232} C_VEL
LIN {X 0,Y 76.931,Z 329.244,A -85,B 0,C 180,E1 -29545.56,E2 -29545.56} C_VEL
LIN {X 0,Y 71.092,Z 340.363,A -85,B 0,C 180,E1 -29548.674,E2 -29548.674} C_VEL
LIN {X 0,Y 64.721,Z 350.669,A -85,B 0,C 180,E1 -29553.035,E2 -29553.035} C_VEL
LIN {X 0,Y 58.421,Z 359.53,A -85,B 0,C 180,E1 -29558.56,E2 -29558.56} C_VEL
LIN {X 0,Y 51.669,Z 368.422,A -85,B 0,C 180,E1 -29567.148,E2 -29567.148} C_VEL
LIN {X 0,Y 46.248,Z 375.497,A -85,B 0,C 180,E1 -29577.868,E2 -29577.868} C_VEL
LIN {X 0,Y 42.795,Z 381.131,A -85,B 0,C 180,E1 -29590.825,E2 -29590.825} C_VEL
LIN {X 0,Y 41.514,Z 385.515,A -85,B 0,C 180,E1 -29605.145,E2 -29605.145} C_VEL
LIN {X 0,Y 41.56,Z 386.735,A -85,B 0,C 180,E1 -29610,E2 -29610} C_VEL
LIN {X 0,Y 41.73,Z 388.716,A -85,B 0,C 180,E1 -29619.696,E2 -29619.696} C_VEL
LIN {X 0,Y 44.93,Z 391.428,A -85,B 0,C 180,E1 -29637.987,E2 -29637.987} C_VEL
LIN {X 0,Y 51.828,Z 392.665,A -85,B 0,C 180,E1 -29652.69,E2 -29652.69} C_VEL
LIN {X 0,Y 61.437,Z 392.418,A -85,B 0,C 180,E1 -29663.204,E2 -29663.204} C_VEL
LIN {X 0,Y 72.59,Z 390.732,A -85,B 0,C 180,E1 -29670.618,E2 -29670.618} C_VEL
LIN {X 0,Y 84.61,Z 387.561,A -85,B 0,C 180,E1 -29676.024,E2 -29676.024} C_VEL
LIN {X 0,Y 94.096,Z 384.117,A -85,B 0,C 180,E1 -29679.009,E2 -29679.009} C_VEL
LIN {X 0,Y 103.822,Z 379.658,A -85,B 0,C 180,E1 -29681.39,E2 -29681.39} C_VEL
LIN {X 0,Y 115.776,Z 372.748,A -85,B 0,C 180,E1 -29683.649,E2 -29683.649} C_VEL
LIN {X 0,Y 118.455,Z 370.994,A -85,B 0,C 180,E1 -29684.076,E2 -29684.076} C_VEL
LIN {X 0,Y 120.978,Z 369.176,A -85,B 0,C 180,E1 -29684.889,E2 -29684.889} C_VEL
LIN {X 0,Y 109.857,Z 376.203,A -85,B 0,C 180,E1 -29686.924,E2 -29686.924} C_VEL
LIN {X 0,Y 100.181,Z 381.096,A -85,B 0,C 180,E1 -29689.158,E2 -29689.158} C_VEL
LIN {X 0,Y 88.596,Z 385.663,A -85,B 0,C 180,E1 -29692.562,E2 -29692.562} C_VEL
LIN {X 0,Y 77.413,Z 388.808,A -85,B 0,C 180,E1 -29697.027,E2 -29697.027} C_VEL
LIN {X 0,Y 69.643,Z 390.282,A -85,B 0,C 180,E1 -29701.168,E2 -29701.168} C_VEL
LIN {X 0,Y 64.622,Z 390.928,A -85,B 0,C 180,E1 -29703.797,E2 -29703.797} C_VEL
LIN {X 0,Y 55.592,Z 391.389,A -85,B 0,C 180,E1 -29707.696,E2 -29707.696} C_VEL
LIN {X 0,Y 48.518,Z 391.181,A -85,B 0,C 180,E1 -29711.693,E2 -29711.693} C_VEL
LIN {X 0,Y 43.907,Z 390.679,A -85,B 0,C 180,E1 -29716.264,E2 -29716.264} C_VEL
LIN {X 0,Y 42.63,Z 390.44,A -85,B 0,C 180,E1 -29718.235,E2 -29718.235} C_VEL
LIN {X 0,Y 35.992,Z 388.017,A -85,B 0,C 180,E1 -29735.86,E2 -29735.86} C_VEL
LIN {X 0,Y 33.676,Z 384.351,A -85,B 0,C 180,E1 -29756.594,E2 -29756.594} C_VEL
LIN {X 0,Y 34.716,Z 380.731,A -85,B 0,C 180,E1 -29772.322,E2 -29772.322} C_VEL
LIN {X 0,Y 38.014,Z 375.824,A -85,B 0,C 180,E1 -29787.351,E2 -29787.351} C_VEL
LIN {X 0,Y 43.962,Z 368.531,A -85,B 0,C 180,E1 -29801.527,E2 -29801.527} C_VEL
LIN {X 0,Y 50.424,Z 360.999,A -85,B 0,C 180,E1 -29810.392,E2 -29810.392} C_VEL
LIN {X 0,Y 57.668,Z 351.849,A -85,B 0,C 180,E1 -29817.195,E2 -29817.195} C_VEL
LIN {X 0,Y 64.639,Z 341.693,A -85,B 0,C 180,E1 -29822.008,E2 -29822.008} C_VEL
LIN {X 0,Y 71.293,Z 330.211,A -85,B 0,C 180,E1 -29825.549,E2 -29825.549} C_VEL
LIN {X 0,Y 76.936,Z 318.118,A -85,B 0,C 180,E1 -29828.069,E2 -29828.069} C_VEL
LIN {X 0,Y 81.686,Z 304.722,A -85,B 0,C 180,E1 -29829.93,E2 -29829.93} C_VEL
LIN {X 0,Y 84.944,Z 291.984,A -85,B 0,C 180,E1 -29831.063,E2 -29831.063} C_VEL
LIN {X 0,Y 87.471,Z 275.999,A -85,B 0,C 180,E1 -29831.801,E2 -29831.801} C_VEL
LIN {X 0,Y 88.642,Z 265.775,A -85,B 0,C 180,E1 -29832.368,E2 -29832.368} C_VEL
LIN {X 0,Y 86.439,Z 259.455,A -85,B 0,C 180,E1 -29836.515,E2 -29836.515} C_VEL
LIN {X 0,Y 84.248,Z 253.886,A -85,B 0,C 180,E1 -29841.3,E2 -29841.3} C_VEL
LIN {X 0,Y 82.241,Z 249.129,A -85,B 0,C 180,E1 -29847.015,E2 -29847.015} C_VEL
LIN {X 0,Y 80.94,Z 246.1,A -85,B 0,C 180,E1 -29852.294,E2 -29852.294} C_VEL
LIN {X 0,Y 79.938,Z 242.753,A -85,B 0,C 180,E1 -29865.263,E2 -29865.263} C_VEL
LIN {X 0,Y 81.009,Z 245.199,A -85,B 0,C 180,E1 -29875.023,E2 -29875.023} C_VEL
LIN {X 0,Y 82.444,Z 249.327,A -85,B 0,C 180,E1 -29881.157,E2 -29881.157} C_VEL
LIN {X 0,Y 84.355,Z 253.921,A -85,B 0,C 180,E1 -29886.464,E2 -29886.464} C_VEL
LIN {X 0,Y 86.74,Z 260.436,A -85,B 0,C 180,E1 -29891.719,E2 -29891.719} C_VEL
LIN {X 0,Y 88.261,Z 265.296,A -85,B 0,C 180,E1 -29894.668,E2 -29894.668} C_VEL
LIN {X 0,Y 88.667,Z 267.401,A -85,B 0,C 180,E1 -29895.544,E2 -29895.544} C_VEL
LIN {X 0,Y 85.536,Z 290.707,A -85,B 0,C 180,E1 -29896.621,E2 -29896.621} C_VEL
LIN {X 0,Y 82.226,Z 304.813,A -85,B 0,C 180,E1 -29897.686,E2 -29897.686} C_VEL
LIN {X 0,Y 78.093,Z 316.915,A -85,B 0,C 180,E1 -29899.099,E2 -29899.099} C_VEL
LIN {X 0,Y 72.585,Z 329.217,A -85,B 0,C 180,E1 -29901.261,E2 -29901.261} C_VEL
LIN {X 0,Y 66.457,Z 340.306,A -85,B 0,C 180,E1 -29904.2,E2 -29904.2} C_VEL
LIN {X 0,Y 59.85,Z 350.358,A -85,B 0,C 180,E1 -29908.3,E2 -29908.3} C_VEL
LIN {X 0,Y 52.93,Z 359.42,A -85,B 0,C 180,E1 -29913.913,E2 -29913.913} C_VEL
LIN {X 0,Y 46.703,Z 366.934,A -85,B 0,C 180,E1 -29921.2,E2 -29921.2} C_VEL
LIN {X 0,Y 40.394,Z 374.272,A -85,B 0,C 180,E1 -29932.486,E2 -29932.486} C_VEL
LIN {X 0,Y 36.156,Z 380.143,A -85,B 0,C 180,E1 -29947.123,E2 -29947.123} C_VEL
LIN {X 0,Y 34.447,Z 384.713,A -85,B 0,C 180,E1 -29964.145,E2 -29964.145} C_VEL
LIN {X 0,Y 34.503,Z 385.948,A -85,B 0,C 180,E1 -29970,E2 -29970} C_VEL
LIN {X 0,Y 34.772,Z 388.046,A -85,B 0,C 180,E1 -29981.661,E2 -29981.661} C_VEL
LIN {X 0,Y 36.193,Z 389.702,A -85,B 0,C 180,E1 -29992.853,E2 -29992.853} C_VEL
LIN {X 0,Y 42.394,Z 391.821,A -85,B 0,C 180,E1 -30011.538,E2 -30011.538} C_VEL
LIN {X 0,Y 51.959,Z 392.525,A -85,B 0,C 180,E1 -30024.249,E2 -30024.249} C_VEL
LIN {X 0,Y 57.457,Z 392.339,A -85,B 0,C 180,E1 -30028.897,E2 -30028.897} C_VEL
LIN {X 0,Y 69.375,Z 390.839,A -85,B 0,C 180,E1 -30035.748,E2 -30035.748} C_VEL
LIN {X 0,Y 81.989,Z 387.886,A -85,B 0,C 180,E1 -30040.548,E2 -30040.548} C_VEL
LIN {X 0,Y 92.735,Z 384.257,A -85,B 0,C 180,E1 -30043.331,E2 -30043.331} C_VEL
LIN {X 0,Y 96.465,Z 382.733,A -85,B 0,C 180,E1 -30044.121,E2 -30044.121} C_VEL
LIN {X 0,Y 98.914,Z 381.673,A -85,B 0,C 180,E1 -30045.105,E2 -30045.105} C_VEL
LIN {X 0,Y 86.154,Z 386.362,A -85,B 0,C 180,E1 -30048.213,E2 -30048.213} C_VEL
LIN {X 0,Y 78.339,Z 388.52,A -85,B 0,C 180,E1 -30050.696,E2 -30050.696} C_VEL
LIN {X 0,Y 65.734,Z 390.726,A -85,B 0,C 180,E1 -30056.198,E2 -30056.198} C_VEL
LIN {X 0,Y 56.27,Z 391.461,A -85,B 0,C 180,E1 -30062.297,E2 -30062.297} C_VEL
LIN {X 0,Y 49.723,Z 391.358,A -85,B 0,C 180,E1 -30068.345,E2 -30068.345} C_VEL
LIN {X 0,Y 42.63,Z 390.44,A -85,B 0,C 180,E1 -30078.235,E2 -30078.235} C_VEL
LIN {X 0,Y 38.808,Z 389.591,A -85,B 0,C 180,E1 -30084.465,E2 -30084.465} C_VEL
LIN {X 0,Y 32.19,Z 387.511,A -85,B 0,C 180,E1 -30095.966,E2 -30095.966} C_VEL
LIN {X 0,Y 28.024,Z 385.316,A -85,B 0,C 180,E1 -30108.267,E2 -30108.267} C_VEL
LIN {X 0,Y 26.675,Z 383.341,A -85,B 0,C 180,E1 -30119.696,E2 -30119.696} C_VEL
LIN {X 0,Y 26.72,Z 382.59,A -85,B 0,C 180,E1 -30123.673,E2 -30123.673} C_VEL
LIN {X 0,Y 29.647,Z 377.74,A -85,B 0,C 180,E1 -30145.15,E2 -30145.15} C_VEL
LIN {X 0,Y 35.119,Z 371.627,A -85,B 0,C 180,E1 -30161.544,E2 -30161.544} C_VEL
LIN {X 0,Y 43.141,Z 363.25,A -85,B 0,C 180,E1 -30174.033,E2 -30174.033} C_VEL
LIN {X 0,Y 51.166,Z 354.158,A -85,B 0,C 180,E1 -30181.402,E2 -30181.402} C_VEL
LIN {X 0,Y 59.09,Z 343.751,A -85,B 0,C 180,E1 -30186.49,E2 -30186.49} C_VEL
LIN {X 0,Y 65.846,Z 333.071,A -85,B 0,C 180,E1 -30189.822,E2 -30189.822} C_VEL
LIN {X 0,Y 71.915,Z 321.306,A -85,B 0,C 180,E1 -30192.212,E2 -30192.212} C_VEL
LIN {X 0,Y 76.631,Z 309.642,A -85,B 0,C 180,E1 -30193.866,E2 -30193.866} C_VEL
LIN {X 0,Y 80.388,Z 297.186,A -85,B 0,C 180,E1 -30195.046,E2 -30195.046} C_VEL
LIN {X 0,Y 83.175,Z 283.526,A -85,B 0,C 180,E1 -30195.72,E2 -30195.72} C_VEL
LIN {X 0,Y 85.126,Z 268.792,A -85,B 0,C 180,E1 -30196.305,E2 -30196.305} C_VEL
LIN {X 0,Y 83.14,Z 262.68,A -85,B 0,C 180,E1 -30200.893,E2 -30200.893} C_VEL
LIN {X 0,Y 81.803,Z 258.852,A -85,B 0,C 180,E1 -30204.649,E2 -30204.649} C_VEL
LIN {X 0,Y 80.396,Z 255.063,A -85,B 0,C 180,E1 -30209.809,E2 -30209.809} C_VEL
LIN {X 0,Y 79.589,Z 252.849,A -85,B 0,C 180,E1 -30213.799,E2 -30213.799} C_VEL
LIN {X 0,Y 78.899,Z 250.008,A -85,B 0,C 180,E1 -30224.5,E2 -30224.5} C_VEL
LIN {X 0,Y 79.008,Z 250.497,A -85,B 0,C 180,E1 -30228.096,E2 -30228.096} C_VEL
LIN {X 0,Y 79.712,Z 252.081,A -85,B 0,C 180,E1 -30233.801,E2 -30233.801} C_VEL
LIN {X 0,Y 80.787,Z 255.751,A -85,B 0,C 180,E1 -30239.283,E2 -30239.283} C_VEL
LIN {X 0,Y 82.241,Z 259.838,A -85,B 0,C 180,E1 -30244.167,E2 -30244.167} C_VEL
LIN {X 0,Y 84.229,Z 266.061,A -85,B 0,C 180,E1 -30249.296,E2 -30249.296} C_VEL
LIN {X 0,Y 85.142,Z 269.417,A -85,B 0,C 180,E1 -30251.454,E2 -30251.454} C_VEL
LIN {X 0,Y 82.155,Z 290.741,A -85,B 0,C 180,E1 -30252.361,E2 -30252.361} C_VEL
LIN {X 0,Y 78.963,Z 303.971,A -85,B 0,C 180,E1 -30253.224,E2 -30253.224} C_VEL
LIN {X 0,Y 74.832,Z 315.943,A -85,B 0,C 180,E1 -30254.412,E2 -30254.412} C_VEL
LIN {X 0,Y 69.509,Z 327.622,A -85,B 0,C 180,E1 -30256.147,E2 -30256.147} C_VEL
LIN {X 0,Y 63.076,Z 338.958,A -85,B 0,C 180,E1 -30258.722,E2 -30258.722} C_VEL
LIN {X 0,Y 56.133,Z 349.148,A -85,B 0,C 180,E1 -30262.351,E2 -30262.351} C_VEL
LIN {X 0,Y 49.307,Z 357.644,A -85,B 0,C 180,E1 -30267.02,E2 -30267.02} C_VEL
LIN {X 0,Y 41.049,Z 366.778,A -85,B 0,C 180,E1 -30275.585,E2 -30275.585} C_VEL
LIN {X 0,Y 33.975,Z 374.091,A -85,B 0,C 180,E1 -30287.755,E2 -30287.755} C_VEL
LIN {X 0,Y 29.745,Z 379.04,A -85,B 0,C 180,E1 -30301.801,E2 -30301.801} C_VEL
LIN {X 0,Y 27.403,Z 383.794,A -85,B 0,C 180,E1 -30322.633,E2 -30322.633} C_VEL
LIN {X 0,Y 27.425,Z 385.121,A -85,B 0,C 180,E1 -30330,E2 -30330} C_VEL
LIN {X 0,Y 27.885,Z 387.31,A -85,B 0,C 180,E1 -30344.598,E2 -30344.598} C_VEL
LIN {X 0,Y 33.072,Z 390.448,A -85,B 0,C 180,E1 -30369.608,E2 -30369.608} C_VEL
LIN {X 0,Y 42.489,Z 392.027,A -85,B 0,C 180,E1 -30385.797,E2 -30385.797} C_VEL
LIN {X 0,Y 54.126,Z 392.195,A -85,B 0,C 180,E1 -30395.357,E2 -30395.357} C_VEL
LIN {X 0,Y 66.77,Z 390.948,A -85,B 0,C 180,E1 -30401.321,E2 -30401.321} C_VEL
LIN {X 0,Y 74.765,Z 389.423,A -85,B 0,C 180,E1 -30403.963,E2 -30403.963} C_VEL
LIN {X 0,Y 77.404,Z 388.814,A -85,B 0,C 180,E1 -30405.33,E2 -30405.33} C_VEL
LIN {X 0,Y 64.269,Z 391.001,A -85,B 0,C 180,E1 -30409.798,E2 -30409.798} C_VEL
LIN {X 0,Y 56.59,Z 391.622,A -85,B 0,C 180,E1 -30413.484,E2 -30413.484} C_VEL
LIN {X 0,Y 47.146,Z 391.574,A -85,B 0,C 180,E1 -30420,E2 -30420} C_VEL
LIN {X 0,Y 37.271,Z 390.368,A -85,B 0,C 180,E1 -30431.586,E2 -30431.586} C_VEL
LIN {X 0,Y 30.34,Z 388.211,A -85,B 0,C 180,E1 -30447.6,E2 -30447.6} C_VEL
LIN {X 0,Y 26.696,Z 384.575,A -85,B 0,C 180,E1 -30472.168,E2 -30472.168} C_VEL
LIN {X 0,Y 26.72,Z 382.59,A -85,B 0,C 180,E1 -30483.673,E2 -30483.673} C_VEL
LIN {X 0,Y 27.054,Z 380.314,A -85,B 0,C 180,E1 -30495.229,E2 -30495.229} C_VEL
LIN {X 0,Y 27.355,Z 377.757,A -85,B 0,C 180,E1 -30506.53,E2 -30506.53} C_VEL
LIN {X 0,Y 30.683,Z 370.8,A -85,B 0,C 180,E1 -30529.836,E2 -30529.836} C_VEL
LIN {X 0,Y 33.95,Z 367.357,A -85,B 0,C 180,E1 -30536.411,E2 -30536.411} C_VEL
LIN {X 0,Y 41.532,Z 360.049,A -85,B 0,C 180,E1 -30544.176,E2 -30544.176} C_VEL
LIN {X 0,Y 49.545,Z 351.154,A -85,B 0,C 180,E1 -30549.668,E2 -30549.668} C_VEL
LIN {X 0,Y 57.59,Z 340.554,A -85,B 0,C 180,E1 -30553.53,E2 -30553.53} C_VEL
LIN {X 0,Y 64.605,Z 329.3,A -85,B 0,C 180,E1 -30556.112,E2 -30556.112} C_VEL
LIN {X 0,Y 70.465,Z 317.415,A -85,B 0,C 180,E1 -30557.886,E2 -30557.886} C_VEL
LIN {X 0,Y 75.222,Z 304.819,A -85,B 0,C 180,E1 -30559.155,E2 -30559.155} C_VEL
LIN {X 0,Y 78.801,Z 291.41,A -85,B 0,C 180,E1 -30560.018,E2 -30560.018} C_VEL
LIN {X 0,Y 81.467,Z 275.074,A -85,B 0,C 180,E1 -30560.513,E2 -30560.513} C_VEL
LIN {X 0,Y 81.876,Z 271.655,A -85,B 0,C 180,E1 -30560.712,E2 -30560.712} C_VEL
LIN {X 0,Y 80.239,Z 265.816,A -85,B 0,C 180,E1 -30565.877,E2 -30565.877} C_VEL
LIN {X 0,Y 79.016,Z 261.856,A -85,B 0,C 180,E1 -30571.046,E2 -30571.046} C_VEL
LIN {X 0,Y 78.267,Z 259.546,A -85,B 0,C 180,E1 -30575.536,E2 -30575.536} C_VEL
LIN {X 0,Y 77.883,Z 257.168,A -85,B 0,C 180,E1 -30584.293,E2 -30584.293} C_VEL
LIN {X 0,Y 77.967,Z 257.518,A -85,B 0,C 180,E1 -30587.599,E2 -30587.599} C_VEL
LIN {X 0,Y 78.454,Z 258.948,A -85,B 0,C 180,E1 -30592.548,E2 -30592.548} C_VEL
LIN {X 0,Y 79.291,Z 262.411,A -85,B 0,C 180,E1 -30597.689,E2 -30597.689} C_VEL
LIN {X 0,Y 80.307,Z 265.942,A -85,B 0,C 180,E1 -30601.919,E2 -30601.919} C_VEL
LIN {X 0,Y 81.834,Z 271.757,A -85,B 0,C 180,E1 -30606.808,E2 -30606.808} C_VEL
LIN {X 0,Y 81.939,Z 272.198,A -85,B 0,C 180,E1 -30607.11,E2 -30607.11} C_VEL
LIN {X 0,Y 79.095,Z 291.327,A -85,B 0,C 180,E1 -30607.818,E2 -30607.818} C_VEL
LIN {X 0,Y 75.61,Z 304.928,A -85,B 0,C 180,E1 -30608.531,E2 -30608.531} C_VEL
LIN {X 0,Y 71.264,Z 316.744,A -85,B 0,C 180,E1 -30609.529,E2 -30609.529} C_VEL
LIN {X 0,Y 65.352,Z 328.984,A -85,B 0,C 180,E1 -30611.095,E2 -30611.095} C_VEL
LIN {X 0,Y 58.672,Z 340.015,A -85,B 0,C 180,E1 -30613.28,E2 -30613.28} C_VEL
LIN {X 0,Y 51.328,Z 350.023,A -85,B 0,C 180,E1 -30616.571,E2 -30616.571} C_VEL
LIN {X 0,Y 43.382,Z 359.067,A -85,B 0,C 180,E1 -30621.327,E2 -30621.327} C_VEL
LIN {X 0,Y 34.475,Z 367.916,A -85,B 0,C 180,E1 -30629.958,E2 -30629.958} C_VEL
LIN {X 0,Y 26.74,Z 374.952,A -85,B 0,C 180,E1 -30643.716,E2 -30643.716} C_VEL
LIN {X 0,Y 22.149,Z 379.725,A -85,B 0,C 180,E1 -30661.579,E2 -30661.579} C_VEL
LIN {X 0,Y 20.36,Z 384.277,A -85,B 0,C 180,E1 -30690,E2 -30690} C_VEL
LIN {X 0,Y 21.11,Z 386.572,A -85,B 0,C 180,E1 -30709.447,E2 -30709.447} C_VEL
LIN {X 0,Y 27.975,Z 389.869,A -85,B 0,C 180,E1 -30738.91,E2 -30738.91} C_VEL
LIN {X 0,Y 38.943,Z 391.691,A -85,B 0,C 180,E1 -30754.468,E2 -30754.468} C_VEL
LIN {X 0,Y 51.568,Z 392.043,A -85,B 0,C 180,E1 -30762.556,E2 -30762.556} C_VEL
LIN {X 0,Y 56.527,Z 391.792,A -85,B 0,C 180,E1 -30765.602,E2 -30765.602} C_VEL
LIN {X 0,Y 45.332,Z 391.779,A -85,B 0,C 180,E1 -30771.082,E2 -30771.082} C_VEL
LIN {X 0,Y 34.871,Z 390.673,A -85,B 0,C 180,E1 -30780.001,E2 -30780.001} C_VEL
LIN {X 0,Y 25.617,Z 388.387,A -85,B 0,C 180,E1 -30795.924,E2 -30795.924} C_VEL
LIN {X 0,Y 19.941,Z 384.724,A -85,B 0,C 180,E1 -30825.18,E2 -30825.18} C_VEL
LIN {X 0,Y 21.302,Z 379.465,A -85,B 0,C 180,E1 -30861.813,E2 -30861.813} C_VEL
LIN {X 0,Y 26.176,Z 374.487,A -85,B 0,C 180,E1 -30881.617,E2 -30881.617} C_VEL
LIN {X 0,Y 33.95,Z 367.357,A -85,B 0,C 180,E1 -30896.411,E2 -30896.411} C_VEL
LIN {X 0,Y 37.362,Z 363.783,A -85,B 0,C 180,E1 -30901.643,E2 -30901.643} C_VEL
LIN {X 0,Y 42.135,Z 357.406,A -85,B 0,C 180,E1 -30910.228,E2 -30910.228} C_VEL
LIN {X 0,Y 47.119,Z 350.442,A -85,B 0,C 180,E1 -30916.787,E2 -30916.787} C_VEL
LIN {X 0,Y 50.561,Z 345.944,A -85,B 0,C 180,E1 -30918.877,E2 -30918.877} C_VEL
LIN {X 0,Y 58.596,Z 334.733,A -85,B 0,C 180,E1 -30921.225,E2 -30921.225} C_VEL
LIN {X 0,Y 65.099,Z 323.321,A -85,B 0,C 180,E1 -30922.768,E2 -30922.768} C_VEL
LIN {X 0,Y 70.514,Z 311.118,A -85,B 0,C 180,E1 -30923.884,E2 -30923.884} C_VEL
LIN {X 0,Y 74.839,Z 297.922,A -85,B 0,C 180,E1 -30924.692,E2 -30924.692} C_VEL
LIN {X 0,Y 77.843,Z 283.858,A -85,B 0,C 180,E1 -30925.102,E2 -30925.102} C_VEL
LIN {X 0,Y 79.118,Z 274.912,A -85,B 0,C 180,E1 -30925.332,E2 -30925.332} C_VEL
LIN {X 0,Y 78.246,Z 270.963,A -85,B 0,C 180,E1 -30929.293,E2 -30929.293} C_VEL
LIN {X 0,Y 77.44,Z 267.92,A -85,B 0,C 180,E1 -30933.712,E2 -30933.712} C_VEL
LIN {X 0,Y 77.046,Z 266.302,A -85,B 0,C 180,E1 -30937.08,E2 -30937.08} C_VEL
LIN {X 0,Y 76.86,Z 264.373,A -85,B 0,C 180,E1 -30944.078,E2 -30944.078} C_VEL
LIN {X 0,Y 76.929,Z 264.548,A -85,B 0,C 180,E1 -30947.071,E2 -30947.071} C_VEL
LIN {X 0,Y 77.224,Z 265.709,A -85,B 0,C 180,E1 -30951.104,E2 -30951.104} C_VEL
LIN {X 0,Y 78.148,Z 270.204,A -85,B 0,C 180,E1 -30957.655,E2 -30957.655} C_VEL
LIN {X 0,Y 79.153,Z 275.122,A -85,B 0,C 180,E1 -30962.41,E2 -30962.41} C_VEL
LIN {X 0,Y 76.635,Z 291.349,A -85,B 0,C 180,E1 -30962.926,E2 -30962.926} C_VEL
LIN {X 0,Y 73.141,Z 304.677,A -85,B 0,C 180,E1 -30963.415,E2 -30963.415} C_VEL
LIN {X 0,Y 68.701,Z 316.499,A -85,B 0,C 180,E1 -30964.124,E2 -30964.124} C_VEL
LIN {X 0,Y 62.634,Z 328.744,A -85,B 0,C 180,E1 -30965.228,E2 -30965.228} C_VEL
LIN {X 0,Y 55.682,Z 339.871,A -85,B 0,C 180,E1 -30966.831,E2 -30966.831} C_VEL
LIN {X 0,Y 48.069,Z 349.795,A -85,B 0,C 180,E1 -30969.283,E2 -30969.283} C_VEL
LIN {X 0,Y 39.664,Z 358.844,A -85,B 0,C 180,E1 -30972.954,E2 -30972.954} C_VEL
LIN {X 0,Y 29.942,Z 367.692,A -85,B 0,C 180,E1 -30980.135,E2 -30980.135} C_VEL
LIN {X 0,Y 21.042,Z 374.732,A -85,B 0,C 180,E1 -30993.386,E2 -30993.386} C_VEL
LIN {X 0,Y 14.541,Z 380.32,A -85,B 0,C 180,E1 -31021.098,E2 -31021.098} C_VEL
LIN {X 0,Y 13.275,Z 383.334,A -85,B 0,C 180,E1 -31050.001,E2 -31050.001} C_VEL
LIN {X 0,Y 14.632,Z 385.765,A -85,B 0,C 180,E1 -31078.707,E2 -31078.707} C_VEL
LIN {X 0,Y 18.537,Z 387.732,A -85,B 0,C 180,E1 -31099.313,E2 -31099.313} C_VEL
LIN {X 0,Y 29.968,Z 390.45,A -85,B 0,C 180,E1 -31119.734,E2 -31119.734} C_VEL
LIN {X 0,Y 36.452,Z 391.281,A -85,B 0,C 180,E1 -31124.584,E2 -31124.584} C_VEL
LIN {X 0,Y 36.24,Z 391.233,A -85,B 0,C 180,E1 -31125.848,E2 -31125.848} C_VEL
LIN {X 0,Y 28.391,Z 389.99,A -85,B 0,C 180,E1 -31131.965,E2 -31131.965} C_VEL
LIN {X 0,Y 17.87,Z 387.054,A -85,B 0,C 180,E1 -31150.514,E2 -31150.514} C_VEL
LIN {X 0,Y 12.475,Z 382.762,A -85,B 0,C 180,E1 -31195.71,E2 -31195.71} C_VEL
LIN {X 0,Y 17.076,Z 377.109,A -85,B 0,C 180,E1 -31241.875,E2 -31241.875} C_VEL
LIN {X 0,Y 24.26,Z 371.519,A -85,B 0,C 180,E1 -31259.646,E2 -31259.646} C_VEL
LIN {X 0,Y 33.028,Z 364.303,A -85,B 0,C 180,E1 -31269.67,E2 -31269.67} C_VEL
LIN {X 0,Y 42.04,Z 355.751,A -85,B 0,C 180,E1 -31275.274,E2 -31275.274} C_VEL
LIN {X 0,Y 50.561,Z 345.944,A -85,B 0,C 180,E1 -31278.877,E2 -31278.877} C_VEL
LIN {X 0,Y 53.844,Z 341.347,A -85,B 0,C 180,E1 -31280.632,E2 -31280.632} C_VEL
LIN {X 0,Y 58.306,Z 333.402,A -85,B 0,C 180,E1 -31284.677,E2 -31284.677} C_VEL
LIN {X 0,Y 62.374,Z 325.053,A -85,B 0,C 180,E1 -31288.129,E2 -31288.129} C_VEL
LIN {X 0,Y 64.864,Z 319.76,A -85,B 0,C 180,E1 -31289.088,E2 -31289.088} C_VEL
LIN {X 0,Y 69.897,Z 307.689,A -85,B 0,C 180,E1 -31289.674,E2 -31289.674} C_VEL
LIN {X 0,Y 74.039,Z 293.818,A -85,B 0,C 180,E1 -31290.111,E2 -31290.111} C_VEL
LIN {X 0,Y 76.584,Z 280.211,A -85,B 0,C 180,E1 -31290.263,E2 -31290.263} C_VEL
LIN {X 0,Y 76.859,Z 278.257,A -85,B 0,C 180,E1 -31290.295,E2 -31290.295} C_VEL
LIN {X 0,Y 76.221,Z 274.828,A -85,B 0,C 180,E1 -31294.775,E2 -31294.775} C_VEL
LIN {X 0,Y 75.874,Z 272.954,A -85,B 0,C 180,E1 -31298.898,E2 -31298.898} C_VEL
LIN {X 0,Y 75.872,Z 271.375,A -85,B 0,C 180,E1 -31304.971,E2 -31304.971} C_VEL
LIN {X 0,Y 76.031,Z 272.334,A -85,B 0,C 180,E1 -31309.346,E2 -31309.346} C_VEL
LIN {X 0,Y 76.663,Z 276.883,A -85,B 0,C 180,E1 -31315.889,E2 -31315.889} C_VEL
LIN {X 0,Y 76.885,Z 278.397,A -85,B 0,C 180,E1 -31317.406,E2 -31317.406} C_VEL
LIN {X 0,Y 74.617,Z 292.077,A -85,B 0,C 180,E1 -31317.752,E2 -31317.752} C_VEL
LIN {X 0,Y 71.016,Z 305.232,A -85,B 0,C 180,E1 -31317.99,E2 -31317.99} C_VEL
LIN {X 0,Y 66.794,Z 316.232,A -85,B 0,C 180,E1 -31318.36,E2 -31318.36} C_VEL
LIN {X 0,Y 60.628,Z 328.463,A -85,B 0,C 180,E1 -31318.912,E2 -31318.912} C_VEL
LIN {X 0,Y 53.093,Z 340.194,A -85,B 0,C 180,E1 -31319.817,E2 -31319.817} C_VEL
LIN {X 0,Y 45.691,Z 349.505,A -85,B 0,C 180,E1 -31321.099,E2 -31321.099} C_VEL
LIN {X 0,Y 36.953,Z 358.553,A -85,B 0,C 180,E1 -31323.143,E2 -31323.143} C_VEL
LIN {X 0,Y 26.578,Z 367.397,A -85,B 0,C 180,E1 -31327.423,E2 -31327.423} C_VEL
LIN {X 0,Y 16.495,Z 374.448,A -85,B 0,C 180,E1 -31336.539,E2 -31336.539} C_VEL
LIN {X 0,Y 9.014,Z 379.211,A -85,B 0,C 180,E1 -31358.77,E2 -31358.77} C_VEL
LIN {X 0,Y 6.206,Z 382.366,A -85,B 0,C 180,E1 -31410.001,E2 -31410.001} C_VEL
LIN {X 0,Y 9.105,Z 384.9,A -85,B 0,C 180,E1 -31460.524,E2 -31460.524} C_VEL
LIN {X 0,Y 14.919,Z 386.978,A -85,B 0,C 180,E1 -31480.418,E2 -31480.418} C_VEL
LIN {X 0,Y 16.096,Z 387.308,A -85,B 0,C 180,E1 -31485.8,E2 -31485.8} C_VEL
LIN {X 0,Y 7.268,Z 383.949,A -85,B 0,C 180,E1 -31514.747,E2 -31514.747} C_VEL
LIN {X 0,Y 9.738,Z 378.217,A -85,B 0,C 180,E1 -31614.615,E2 -31614.615} C_VEL
LIN {X 0,Y 19.629,Z 371.956,A -85,B 0,C 180,E1 -31634.266,E2 -31634.266} C_VEL
LIN {X 0,Y 29.346,Z 364.739,A -85,B 0,C 180,E1 -31641.108,E2 -31641.108} C_VEL
LIN {X 0,Y 38.878,Z 356.252,A -85,B 0,C 180,E1 -31644.437,E2 -31644.437} C_VEL
LIN {X 0,Y 47.406,Z 346.944,A -85,B 0,C 180,E1 -31646.504,E2 -31646.504} C_VEL
LIN {X 0,Y 55.311,Z 336.434,A -85,B 0,C 180,E1 -31647.8,E2 -31647.8} C_VEL
LIN {X 0,Y 61.699,Z 325.952,A -85,B 0,C 180,E1 -31648.684,E2 -31648.684} C_VEL
LIN {X 0,Y 64.864,Z 319.76,A -85,B 0,C 180,E1 -31649.088,E2 -31649.088} C_VEL
LIN {X 0,Y 66.364,Z 316.164,A -85,B 0,C 180,E1 -31649.869,E2 -31649.869} C_VEL
LIN {X 0,Y 68.144,Z 310.42,A -85,B 0,C 180,E1 -31652.518,E2 -31652.518} C_VEL
LIN {X 0,Y 69.802,Z 304.564,A -85,B 0,C 180,E1 -31654.958,E2 -31654.958} C_VEL
LIN {X 0,Y 70.884,Z 300.796,A -85,B 0,C 180,E1 -31655.517,E2 -31655.517} C_VEL
LIN {X 0,Y 74.058,Z 287.899,A -85,B 0,C 180,E1 -31655.56,E2 -31655.56} C_VEL
LIN {X 0,Y 75.02,Z 282.138,A -85,B 0,C 180,E1 -31655.594,E2 -31655.594} C_VEL
LIN {X 0,Y 74.822,Z 279.93,A -85,B 0,C 180,E1 -31659.533,E2 -31659.533} C_VEL
LIN {X 0,Y 74.881,Z 278.526,A -85,B 0,C 180,E1 -31665.882,E2 -31665.882} C_VEL
LIN {X 0,Y 74.916,Z 279.451,A -85,B 0,C 180,E1 -31668.4,E2 -31668.4} C_VEL
LIN {X 0,Y 75.078,Z 282.09,A -85,B 0,C 180,E1 -31672.254,E2 -31672.254} C_VEL
LIN {X 0,Y 72.516,Z 295.318,A -85,B 0,C 180,E1 -31672.361,E2 -31672.361} C_VEL
LIN {X 0,Y 68.308,Z 308.989,A -85,B 0,C 180,E1 -31672.351,E2 -31672.351} C_VEL
LIN {X 0,Y 62.938,Z 321.413,A -85,B 0,C 180,E1 -31672.321,E2 -31672.321} C_VEL
LIN {X 0,Y 55.884,Z 333.811,A -85,B 0,C 180,E1 -31672.173,E2 -31672.173} C_VEL
LIN {X 0,Y 48.767,Z 343.831,A -85,B 0,C 180,E1 -31672.222,E2 -31672.222} C_VEL
LIN {X 0,Y 40.786,Z 353.021,A -85,B 0,C 180,E1 -31672.231,E2 -31672.231} C_VEL
LIN {X 0,Y 30.15,Z 362.902,A -85,B 0,C 180,E1 -31672.175,E2 -31672.175} C_VEL
LIN {X 0,Y 19.535,Z 370.82,A -85,B 0,C 180,E1 -31671.628,E2 -31671.628} C_VEL
LIN {X 0,Y 8.93,Z 377.136,A -85,B 0,C 180,E1 -31669.672,E2 -31669.672} C_VEL
LIN {X 0,Y 7.172,Z 378.033,A -85,B 0,C 180,E1 -31668.482,E2 -31668.482} C_VEL
LIN {X 0,Y 7.422,Z 377.875,A -85,B 0,C 180,E1 -31661.25,E2 -31661.25} C_VEL
LIN {X 0,Y 17.011,Z 372.337,A -85,B 0,C 180,E1 -31655.597,E2 -31655.597} C_VEL
LIN {X 0,Y 27.122,Z 365.176,A -85,B 0,C 180,E1 -31655.085,E2 -31655.085} C_VEL
LIN {X 0,Y 37.108,Z 356.505,A -85,B 0,C 180,E1 -31654.894,E2 -31654.894} C_VEL
LIN {X 0,Y 46.498,Z 346.335,A -85,B 0,C 180,E1 -31655.079,E2 -31655.079} C_VEL
LIN {X 0,Y 54.226,Z 336.044,A -85,B 0,C 180,E1 -31655.127,E2 -31655.127} C_VEL
LIN {X 0,Y 60.954,Z 324.943,A -85,B 0,C 180,E1 -31655.23,E2 -31655.23} C_VEL
LIN {X 0,Y 66.718,Z 312.642,A -85,B 0,C 180,E1 -31655.374,E2 -31655.374} C_VEL
LIN {X 0,Y 70.884,Z 300.796,A -85,B 0,C 180,E1 -31655.517,E2 -31655.517} C_VEL
LIN {X 0,Y 70.864,Z 300.55,A -85,B 0,C 180,E1 -31656.148,E2 -31656.148} C_VEL
LIN {X 0,Y 70.31,Z 301.703,A -85,B 0,C 180,E1 -31657.733,E2 -31657.733} C_VEL
LIN {X 0,Y 68.942,Z 305.357,A -85,B 0,C 180,E1 -31660.178,E2 -31660.178} C_VEL
LIN {X 0,Y 65.592,Z 314.016,A -85,B 0,C 180,E1 -31663.56,E2 -31663.56} C_VEL
LIN {X 0,Y 63.43,Z 318.966,A -85,B 0,C 180,E1 -31664.949,E2 -31664.949} C_VEL
LIN {X 0,Y 61.012,Z 323.92,A -85,B 0,C 180,E1 -31665.586,E2 -31665.586} C_VEL
LIN {X 0,Y 59.686,Z 326.359,A -85,B 0,C 180,E1 -31665.513,E2 -31665.513} C_VEL
LIN {X 0,Y 52.853,Z 337.42,A -85,B 0,C 180,E1 -31664.577,E2 -31664.577} C_VEL
LIN {X 0,Y 49.574,Z 341.97,A -85,B 0,C 180,E1 -31664.05,E2 -31664.05} C_VEL
LIN {X 0,Y 49.095,Z 342.604,A -85,B 0,C 180,E1 -31663.363,E2 -31663.363} C_VEL
LIN {X 0,Y 56.234,Z 332.227,A -85,B 0,C 180,E1 -31662.357,E2 -31662.357} C_VEL
LIN {X 0,Y 62.915,Z 320.067,A -85,B 0,C 180,E1 -31661.715,E2 -31661.715} C_VEL
LIN {X 0,Y 67.966,Z 307.954,A -85,B 0,C 180,E1 -31661.397,E2 -31661.397} C_VEL
LIN {X 0,Y 72.004,Z 294.552,A -85,B 0,C 180,E1 -31661.157,E2 -31661.157} C_VEL
LIN {X 0,Y 73.633,Z 286.884,A -85,B 0,C 180,E1 -31661.029,E2 -31661.029} C_VEL
LIN {X 0,Y 73.799,Z 285.618,A -85,B 0,C 180,E1 -31665.671,E2 -31665.671} C_VEL
LIN {X 0,Y 73.755,Z 286.188,A -85,B 0,C 180,E1 -31666.768,E2 -31666.768} C_VEL
LIN {X 0,Y 71.027,Z 298.465,A -85,B 0,C 180,E1 -31666.666,E2 -31666.666} C_VEL
LIN {X 0,Y 66.654,Z 311.515,A -85,B 0,C 180,E1 -31666.333,E2 -31666.333} C_VEL
LIN {X 0,Y 60.762,Z 324.374,A -85,B 0,C 180,E1 -31665.626,E2 -31665.626} C_VEL
LIN {X 0,Y 59.686,Z 326.359,A -85,B 0,C 180,E1 -31665.513,E2 -31665.513} C_VEL
LIN {X 0,Y 59.425,Z 327.355,A -85,B 0,C 180,E1 -31665.468,E2 -31665.468} C_VEL
LIN {X 0,Y 59.425,Z 600,A -85,B 0,C 180,E1 -31665.468,E2 -31665.468} C_VEL
LIN {X 0,Y 59.425,Z 600,A -85,B 0,C 180,E1 -31665.468,E2 -31665.468}

QRS_NEXT_CUT()

QRS_NEXT()
QRS_HOME()

END
